(* CoDeSys 2.3 export: CRYNKAMOGILEV.EXP *)
(* Libraries: Iecsfc.lib 30.1.13 14:05:12, Standard.lib 20.5.14 09:13:26, SYSLIBCALLBACK.LIB 30.1.13 14:05:12, SysLibRtc.lib 30.1.13 14:05:12, SysLibTime.lib 30.1.13 14:05:12, Util_no_Real.lib 30.1.13 14:05:12 *)

(* PLC configuration (modules and I/O channels)
PLC Configuration [Root] node -1, in %IB0 out %QB0
  K-Bus [K_Bus] node 0, in %IB0 out %QB0 {param 201019000 = 1; param 201019001 = 10000; param 201019002 = 0; param 201019003 = 1}
    0750-1405 16 DI 24V DC 3.0ms [Type_1_16_Channels] node 0, in %IB56 out %QB16
      _Pump_FeedbackOn_1 AT %IX28.0 [BOOLOnX_I] Ch_1 Digital input
      _Pump_Alm_1 AT %IX28.1 [BOOLOnX_I] Ch_2 Digital input
      _Pump_FeedbackOn_2 AT %IX28.2 [BOOLOnX_I] Ch_3 Digital input
      _Pump_Alm_2 AT %IX28.3 [BOOLOnX_I] Ch_4 Digital input
      _Pump_FeedbackOn_3 AT %IX28.4 [BOOLOnX_I] Ch_5 Digital input
      _Pump_Alm_3 AT %IX28.5 [BOOLOnX_I] Ch_6 Digital input
      _Pump_FeedbackOn_4 AT %IX28.6 [BOOLOnX_I] Ch_7 Digital input
      _Pump_Alm_4 AT %IX28.7 [BOOLOnX_I] Ch_8 Digital input
      _DI_FeedBackSwitchLine1 AT %IX28.8 [BOOLOnX_I] Ch_9 Digital input
      _DI_FeedBackSwitchLine2 AT %IX28.9 [BOOLOnX_I] Ch_10 Digital input
      _DI_FeedBackSwitchLine3 AT %IX28.10 [BOOLOnX_I] Ch_11 Digital input
      _DI_FeedBackSwitchLine4 AT %IX28.11 [BOOLOnX_I] Ch_12 Digital input
      _LH_1 AT %IX28.12 [BOOLOnX_I] Ch_13 Digital input
      _LH_2 AT %IX28.13 [BOOLOnX_I] Ch_14 Digital input
      _LH_3 AT %IX28.14 [BOOLOnX_I] Ch_15 Digital input
      _LH_4 AT %IX28.15 [BOOLOnX_I] Ch_16 Digital input
    0750-1405 16 DI 24V DC 3.0ms [Type_1_16_Channels] node 1, in %IB56 out %QB16
      _FC_1 AT %IX29.0 [BOOLOnX_I] Ch_1 Digital input
      _FC_2 AT %IX29.1 [BOOLOnX_I] Ch_2 Digital input
      _FC_3 AT %IX29.2 [BOOLOnX_I] Ch_3 Digital input
      _FC_4 AT %IX29.3 [BOOLOnX_I] Ch_4 Digital input
      _Permition_Line_1 AT %IX29.4 [BOOLOnX_I] Ch_5 Digital input
      _Permition_Line_2 AT %IX29.5 [BOOLOnX_I] Ch_6 Digital input
      _Permition_Line_3 AT %IX29.6 [BOOLOnX_I] Ch_7 Digital input
      _Permition_Line_4 AT %IX29.7 [BOOLOnX_I] Ch_8 Digital input
      _Permition_Line_5 AT %IX29.8 [BOOLOnX_I] Ch_9 Digital input
      AT %IX29.9 [BOOLOnX_I] Ch_10 Digital input
      AT %IX29.10 [BOOLOnX_I] Ch_11 Digital input
      AT %IX29.11 [BOOLOnX_I] Ch_12 Digital input
      AT %IX29.12 [BOOLOnX_I] Ch_13 Digital input
      AT %IX29.13 [BOOLOnX_I] Ch_14 Digital input
      AT %IX29.14 [BOOLOnX_I] Ch_15 Digital input
      AT %IX29.15 [BOOLOnX_I] Ch_16 Digital input
    0750-1405 16 DI 24V DC 3.0ms [Type_1_16_Channels] node 2, in %IB58 out %QB16
      AT %IX30.0 [BOOLOnX_I] Ch_1 Digital input
      AT %IX30.1 [BOOLOnX_I] Ch_2 Digital input
      AT %IX30.2 [BOOLOnX_I] Ch_3 Digital input
      AT %IX30.3 [BOOLOnX_I] Ch_4 Digital input
      AT %IX30.4 [BOOLOnX_I] Ch_5 Digital input
      AT %IX30.5 [BOOLOnX_I] Ch_6 Digital input
      AT %IX30.6 [BOOLOnX_I] Ch_7 Digital input
      AT %IX30.7 [BOOLOnX_I] Ch_8 Digital input
      _DI_V101 AT %IX30.8 [BOOLOnX_I] Ch_9 Digital input
      _DI_V102 AT %IX30.9 [BOOLOnX_I] Ch_10 Digital input
      _DI_V103 AT %IX30.10 [BOOLOnX_I] Ch_11 Digital input
      _DI_V104 AT %IX30.11 [BOOLOnX_I] Ch_12 Digital input
      _DI_V105 AT %IX30.12 [BOOLOnX_I] Ch_13 Digital input
      _DI_V106 AT %IX30.13 [BOOLOnX_I] Ch_14 Digital input
      _DI_V107 AT %IX30.14 [BOOLOnX_I] Ch_15 Digital input
      _DI_V108 AT %IX30.15 [BOOLOnX_I] Ch_16 Digital input
    0750-1405 16 DI 24V DC 3.0ms [Type_1_16_Channels] node 3, in %IB60 out %QB16
      _DI_V109 AT %IX31.0 [BOOLOnX_I] Ch_1 Digital input
      _DI_V110 AT %IX31.1 [BOOLOnX_I] Ch_2 Digital input
      _DI_V111 AT %IX31.2 [BOOLOnX_I] Ch_3 Digital input
      _DI_V201 AT %IX31.3 [BOOLOnX_I] Ch_4 Digital input
      _DI_V202 AT %IX31.4 [BOOLOnX_I] Ch_5 Digital input
      _DI_V203 AT %IX31.5 [BOOLOnX_I] Ch_6 Digital input
      _DI_V204 AT %IX31.6 [BOOLOnX_I] Ch_7 Digital input
      _DI_V205 AT %IX31.7 [BOOLOnX_I] Ch_8 Digital input
      _DI_V206 AT %IX31.8 [BOOLOnX_I] Ch_9 Digital input
      _DI_V207 AT %IX31.9 [BOOLOnX_I] Ch_10 Digital input
      _DI_V208 AT %IX31.10 [BOOLOnX_I] Ch_11 Digital input
      _DI_V209 AT %IX31.11 [BOOLOnX_I] Ch_12 Digital input
      _DI_V210 AT %IX31.12 [BOOLOnX_I] Ch_13 Digital input
      _DI_V211 AT %IX31.13 [BOOLOnX_I] Ch_14 Digital input
      _DI_V301 AT %IX31.14 [BOOLOnX_I] Ch_15 Digital input
      _DI_V302 AT %IX31.15 [BOOLOnX_I] Ch_16 Digital input
    0750-1405 16 DI 24V DC 3.0ms [Type_1_16_Channels] node 4, in %IB62 out %QB16
      _DI_V303 AT %IX32.0 [BOOLOnX_I] Ch_1 Digital input
      _DI_V304 AT %IX32.1 [BOOLOnX_I] Ch_2 Digital input
      _DI_V305 AT %IX32.2 [BOOLOnX_I] Ch_3 Digital input
      _DI_V306 AT %IX32.3 [BOOLOnX_I] Ch_4 Digital input
      _DI_V307 AT %IX32.4 [BOOLOnX_I] Ch_5 Digital input
      _DI_V308 AT %IX32.5 [BOOLOnX_I] Ch_6 Digital input
      _DI_V309 AT %IX32.6 [BOOLOnX_I] Ch_7 Digital input
      _DI_V310 AT %IX32.7 [BOOLOnX_I] Ch_8 Digital input
      _DI_V311 AT %IX32.8 [BOOLOnX_I] Ch_9 Digital input
      _DI_V401 AT %IX32.9 [BOOLOnX_I] Ch_10 Digital input
      _DI_V402 AT %IX32.10 [BOOLOnX_I] Ch_11 Digital input
      _DI_V403 AT %IX32.11 [BOOLOnX_I] Ch_12 Digital input
      _DI_V404 AT %IX32.12 [BOOLOnX_I] Ch_13 Digital input
      _DI_V405 AT %IX32.13 [BOOLOnX_I] Ch_14 Digital input
      _DI_V406 AT %IX32.14 [BOOLOnX_I] Ch_15 Digital input
      _DI_V407 AT %IX32.15 [BOOLOnX_I] Ch_16 Digital input
    0750-1405 16 DI 24V DC 3.0ms [Type_1_16_Channels] node 5, in %IB64 out %QB16
      _DI_V408 AT %IX33.0 [BOOLOnX_I] Ch_1 Digital input
      _DI_V409 AT %IX33.1 [BOOLOnX_I] Ch_2 Digital input
      _DI_V410 AT %IX33.2 [BOOLOnX_I] Ch_3 Digital input
      _DI_V411 AT %IX33.3 [BOOLOnX_I] Ch_4 Digital input
      _DI_V510 AT %IX33.4 [BOOLOnX_I] Ch_5 Digital input
      _DI_V511 AT %IX33.5 [BOOLOnX_I] Ch_6 Digital input
      _DI_V512 AT %IX33.6 [BOOLOnX_I] Ch_7 Digital input
      _DI_V513 AT %IX33.7 [BOOLOnX_I] Ch_8 Digital input
      _DI_V514 AT %IX33.8 [BOOLOnX_I] Ch_9 Digital input
      _DI_V515 AT %IX33.9 [BOOLOnX_I] Ch_10 Digital input
      _DI_V501 AT %IX33.10 [BOOLOnX_I] Ch_11 Digital input
      AT %IX33.11 [BOOLOnX_I] Ch_12 Digital input
      AT %IX33.12 [BOOLOnX_I] Ch_13 Digital input
      AT %IX33.13 [BOOLOnX_I] Ch_14 Digital input
      AT %IX33.14 [BOOLOnX_I] Ch_15 Digital input
      AT %IX33.15 [BOOLOnX_I] Ch_16 Digital input
    0750-1504 16 DO 24V DC 0.5A [Type_10_16_Channels] node 6, in %IB66 out %QB16
      _DO_PumpOn_1 AT %QX8.0 [BOOLOnX_Q] Ch_1 Digital output
      _DO_PumpOn_2 AT %QX8.1 [BOOLOnX_Q] Ch_2 Digital output
      _DO_PumpOn_3 AT %QX8.2 [BOOLOnX_Q] Ch_3 Digital output
      _DO_PumpOn_4 AT %QX8.3 [BOOLOnX_Q] Ch_4 Digital output
      _HL_Green AT %QX8.4 [BOOLOnX_Q] Ch_5 Digital output
      _HL_Yellow AT %QX8.5 [BOOLOnX_Q] Ch_6 Digital output
      _HL_Red AT %QX8.6 [BOOLOnX_Q] Ch_7 Digital output
      _Alm AT %QX8.7 [BOOLOnX_Q] Ch_8 Digital output
      _Ready_Line_1 AT %QX8.8 [BOOLOnX_Q] Ch_9 Digital output
      _Working_Line_1 AT %QX8.9 [BOOLOnX_Q] Ch_10 Digital output
      _Working_Pump_1 AT %QX8.10 [BOOLOnX_Q] Ch_11 Digital output
      _SwitchOnRemotePump_1 AT %QX8.11 [BOOLOnX_Q] Ch_12 Digital output
      _SwitchOnRemotePump_2 AT %QX8.12 [BOOLOnX_Q] Ch_13 Digital output
      _Ready_Line_2 AT %QX8.13 [BOOLOnX_Q] Ch_14 Digital output
      _Working_Line_2 AT %QX8.14 [BOOLOnX_Q] Ch_15 Digital output
      _Working_Pump_2 AT %QX8.15 [BOOLOnX_Q] Ch_16 Digital output
    0750-1504 16 DO 24V DC 0.5A [Type_10_16_Channels] node 7, in %IB68 out %QB16
      AT %QX9.0 [BOOLOnX_Q] Ch_1 Digital output
      AT %QX9.1 [BOOLOnX_Q] Ch_2 Digital output
      _Ready_Line_3 AT %QX9.2 [BOOLOnX_Q] Ch_3 Digital output
      _Working_Line_3 AT %QX9.3 [BOOLOnX_Q] Ch_4 Digital output
      _Working_Pump_3 AT %QX9.4 [BOOLOnX_Q] Ch_5 Digital output
      _SwitchOnRemotePump_3 AT %QX9.5 [BOOLOnX_Q] Ch_6 Digital output
      AT %QX9.6 [BOOLOnX_Q] Ch_7 Digital output
      _Ready_Line_4 AT %QX9.7 [BOOLOnX_Q] Ch_8 Digital output
      _Working_Line_4 AT %QX9.8 [BOOLOnX_Q] Ch_9 Digital output
      _Working_Pump_4 AT %QX9.9 [BOOLOnX_Q] Ch_10 Digital output
      _SwitchOnRemotePump_4 AT %QX9.10 [BOOLOnX_Q] Ch_11 Digital output
      AT %QX9.11 [BOOLOnX_Q] Ch_12 Digital output
      AT %QX9.12 [BOOLOnX_Q] Ch_13 Digital output
      AT %QX9.13 [BOOLOnX_Q] Ch_14 Digital output
      AT %QX9.14 [BOOLOnX_Q] Ch_15 Digital output
      AT %QX9.15 [BOOLOnX_Q] Ch_16 Digital output
    0750-1504 16 DO 24V DC 0.5A [Type_10_16_Channels] node 8, in %IB68 out %QB18
      _DO_V101 AT %QX10.0 [BOOLOnX_Q] Ch_1 Digital output
      _DO_V102 AT %QX10.1 [BOOLOnX_Q] Ch_2 Digital output
      _DO_V103 AT %QX10.2 [BOOLOnX_Q] Ch_3 Digital output
      _DO_V104 AT %QX10.3 [BOOLOnX_Q] Ch_4 Digital output
      _DO_V105 AT %QX10.4 [BOOLOnX_Q] Ch_5 Digital output
      _DO_V106 AT %QX10.5 [BOOLOnX_Q] Ch_6 Digital output
      _DO_V107 AT %QX10.6 [BOOLOnX_Q] Ch_7 Digital output
      _DO_V108 AT %QX10.7 [BOOLOnX_Q] Ch_8 Digital output
      _DO_V109 AT %QX10.8 [BOOLOnX_Q] Ch_9 Digital output
      _DO_V110 AT %QX10.9 [BOOLOnX_Q] Ch_10 Digital output
      _DO_V111 AT %QX10.10 [BOOLOnX_Q] Ch_11 Digital output
      _DO_V201 AT %QX10.11 [BOOLOnX_Q] Ch_12 Digital output
      _DO_V202 AT %QX10.12 [BOOLOnX_Q] Ch_13 Digital output
      _DO_V203 AT %QX10.13 [BOOLOnX_Q] Ch_14 Digital output
      _DO_V204 AT %QX10.14 [BOOLOnX_Q] Ch_15 Digital output
      _DO_V205 AT %QX10.15 [BOOLOnX_Q] Ch_16 Digital output
    0750-1504 16 DO 24V DC 0.5A [Type_10_16_Channels] node 9, in %IB68 out %QB20
      _DO_V206 AT %QX11.0 [BOOLOnX_Q] Ch_1 Digital output
      _DO_V207 AT %QX11.1 [BOOLOnX_Q] Ch_2 Digital output
      _DO_V208 AT %QX11.2 [BOOLOnX_Q] Ch_3 Digital output
      _DO_V209 AT %QX11.3 [BOOLOnX_Q] Ch_4 Digital output
      _DO_V210 AT %QX11.4 [BOOLOnX_Q] Ch_5 Digital output
      _DO_V211 AT %QX11.5 [BOOLOnX_Q] Ch_6 Digital output
      _DO_V301 AT %QX11.6 [BOOLOnX_Q] Ch_7 Digital output
      _DO_V302 AT %QX11.7 [BOOLOnX_Q] Ch_8 Digital output
      _DO_V303 AT %QX11.8 [BOOLOnX_Q] Ch_9 Digital output
      _DO_V304 AT %QX11.9 [BOOLOnX_Q] Ch_10 Digital output
      _DO_V305 AT %QX11.10 [BOOLOnX_Q] Ch_11 Digital output
      _DO_V306 AT %QX11.11 [BOOLOnX_Q] Ch_12 Digital output
      AT %QX11.12 [BOOLOnX_Q] Ch_13 Digital output
      _DO_PA1 AT %QX11.13 [BOOLOnX_Q] Ch_14 Digital output
      _DO_PA2 AT %QX11.14 [BOOLOnX_Q] Ch_15 Digital output
      _DO_PA3 AT %QX11.15 [BOOLOnX_Q] Ch_16 Digital output
    0750-1504 16 DO 24V DC 0.5A [Type_10_16_Channels] node 10, in %IB68 out %QB22
      _DO_V308 AT %QX12.0 [BOOLOnX_Q] Ch_1 Digital output
      _DO_V309 AT %QX12.1 [BOOLOnX_Q] Ch_2 Digital output
      _DO_V310 AT %QX12.2 [BOOLOnX_Q] Ch_3 Digital output
      _DO_V311 AT %QX12.3 [BOOLOnX_Q] Ch_4 Digital output
      _DO_V401 AT %QX12.4 [BOOLOnX_Q] Ch_5 Digital output
      _DO_V402 AT %QX12.5 [BOOLOnX_Q] Ch_6 Digital output
      _DO_V403 AT %QX12.6 [BOOLOnX_Q] Ch_7 Digital output
      _DO_V404 AT %QX12.7 [BOOLOnX_Q] Ch_8 Digital output
      _DO_V405 AT %QX12.8 [BOOLOnX_Q] Ch_9 Digital output
      _DO_V406 AT %QX12.9 [BOOLOnX_Q] Ch_10 Digital output
      _DO_V407 AT %QX12.10 [BOOLOnX_Q] Ch_11 Digital output
      _DO_V408 AT %QX12.11 [BOOLOnX_Q] Ch_12 Digital output
      _DO_V409 AT %QX12.12 [BOOLOnX_Q] Ch_13 Digital output
      _DO_V410 AT %QX12.13 [BOOLOnX_Q] Ch_14 Digital output
      _DO_V411 AT %QX12.14 [BOOLOnX_Q] Ch_15 Digital output
      _DO_V510 AT %QX12.15 [BOOLOnX_Q] Ch_16 Digital output
    0750-1504 16 DO 24V DC 0.5A [Type_10_16_Channels] node 11, in %IB68 out %QB24
      _DO_V511 AT %QX13.0 [BOOLOnX_Q] Ch_1 Digital output
      _DO_V512 AT %QX13.1 [BOOLOnX_Q] Ch_2 Digital output
      _DO_V513 AT %QX13.2 [BOOLOnX_Q] Ch_3 Digital output
      _DO_V514 AT %QX13.3 [BOOLOnX_Q] Ch_4 Digital output
      _DO_V515 AT %QX13.4 [BOOLOnX_Q] Ch_5 Digital output
      _DO_V501 AT %QX13.5 [BOOLOnX_Q] Ch_6 Digital output
      _DO_V307 AT %QX13.6 [BOOLOnX_Q] Ch_7 Digital output
      AT %QX13.7 [BOOLOnX_Q] Ch_8 Digital output
      AT %QX13.8 [BOOLOnX_Q] Ch_9 Digital output
      AT %QX13.9 [BOOLOnX_Q] Ch_10 Digital output
      AT %QX13.10 [BOOLOnX_Q] Ch_11 Digital output
      AT %QX13.11 [BOOLOnX_Q] Ch_12 Digital output
      _DO_PA4 AT %QX13.12 [BOOLOnX_Q] Ch_13 Digital output
      _DO_PA11 AT %QX13.13 [BOOLOnX_Q] Ch_14 Digital output
      _DO_PA12 AT %QX13.14 [BOOLOnX_Q] Ch_15 Digital output
      AT %QX13.15 [BOOLOnX_Q] Ch_16 Digital output
    0750-0496 8AI 0-20mA/4-20mA S.E. [Type_63_8_Channels] node 12, in %IB56 out %QB8
      _AI_Conc_Line1 AT %IW0 [INTOnW_I] Ch_1 signed Input value
      _AI_Conc_Line2 AT %IW1 [INTOnW_I] Ch_2 signed Input value
      _AI_Conc_Line3 AT %IW2 [INTOnW_I] Ch_3 signed Input value
      _AI_Conc_Line4 AT %IW3 [INTOnW_I] Ch_4 signed Input value
      _AI_AccidLevel AT %IW4 [INTOnW_I] Ch_5 signed Input value
      _AI_AlkaliLevel AT %IW5 [INTOnW_I] Ch_6 signed Input value
      _AI_CleanWaterLevel AT %IW6 [INTOnW_I] Ch_7 signed Input value
      _AI_UsedWaterLevel AT %IW7 [INTOnW_I] Ch_8 signed Input value
    0750-0496 8AI 0-20mA/4-20mA S.E. [Type_63_8_Channels] node 13, in %IB56 out %QB8
      _AI_Flaw_Line1 AT %IW8 [INTOnW_I] Ch_1 signed Input value
      _AI_Flaw_Line2 AT %IW9 [INTOnW_I] Ch_2 signed Input value
      _AI_Flaw_Line3 AT %IW10 [INTOnW_I] Ch_3 signed Input value
      _AI_Flaw_Line4 AT %IW11 [INTOnW_I] Ch_4 signed Input value
      AT %IW12 [INTOnW_I] Ch_5 signed Input value
      AT %IW13 [INTOnW_I] Ch_6 signed Input value
      AT %IW14 [INTOnW_I] Ch_7 signed Input value
      AT %IW15 [INTOnW_I] Ch_8 signed Input value
    0750-0450 4AI RTD/ adj. [Type_62_4_Channels] node 14, in %IB72 out %QB8
      _AI_Heater_BackTget_1 AT %IW16 [INTOnW_I] Ch_1 signed Input value
      _AI_Heater_BackTget_2 AT %IW17 [INTOnW_I] Ch_2 signed Input value
      _AI_Heater_BackTget_3 AT %IW18 [INTOnW_I] Ch_3 signed Input value
      _AI_Heater_BackTget_4 AT %IW19 [INTOnW_I] Ch_4 signed Input value
    0750-0450 4AI RTD/ adj. [Type_62_4_Channels] node 15, in %IB88 out %QB8
      _AI_Heater_Tget_1 AT %IW20 [INTOnW_I] Ch_1 signed Input value
      _AI_Heater_Tget_2 AT %IW21 [INTOnW_I] Ch_2 signed Input value
      _AI_Heater_Tget_3 AT %IW22 [INTOnW_I] Ch_3 signed Input value
      _AI_Heater_Tget_4 AT %IW23 [INTOnW_I] Ch_4 signed Input value
    0750-0450 4AI RTD/ adj. [Type_62_4_Channels] node 16, in %IB96 out %QB8
      _AI_Temp_Accid AT %IW24 [INTOnW_I] Ch_1 signed Input value
      _AI_Temp_Alkali AT %IW25 [INTOnW_I] Ch_2 signed Input value
      AT %IW26 [INTOnW_I] Ch_3 signed Input value
      AT %IW27 [INTOnW_I] Ch_4 signed Input value
    0750-0555 4 AO 4-20mA [Type_14_4_Channels] node 17, in %IB104 out %QB8
      _AO_PumpSpeedSet_1 AT %QW0 [WORDOnW_Q] Ch_1 Analog output
      _AO_PumpSpeedSet_2 AT %QW1 [WORDOnW_Q] Ch_2 Analog output
      _AO_PumpSpeedSet_3 AT %QW2 [WORDOnW_Q] Ch_3 Analog output
      _AO_PumpSpeedSet_4 AT %QW3 [WORDOnW_Q] Ch_4 Analog output
    0750-0555 4 AO 4-20mA [Type_14_4_Channels] node 18, in %IB112 out %QB8
      _AO_HeaterPowerSet_1 AT %QW4 [WORDOnW_Q] Ch_1 Analog output
      _AO_HeaterPowerSet_2 AT %QW5 [WORDOnW_Q] Ch_2 Analog output
      _AO_HeaterPowerSet_3 AT %QW6 [WORDOnW_Q] Ch_3 Analog output
      _AO_HeaterPowerSet_4 AT %QW7 [WORDOnW_Q] Ch_4 Analog output
  Modbus variables [PFC200MODBUS] node 1, in %IB0 out %QB0 {param 2010330101 = 1; param 2010330102 = 1; param 2010330201 = 1; param 2010330202 = 502; param 2010330203 = 600; param 2010330301 = 1; param 2010330302 = 502; param 2010330401 = 0; param 2010330402 = 1; param 2010330403 = 5000; param 2010330404 = 0; param 2010330405 = 115200; param 2010330406 = 1; param 2010330407 = 1; param 2010330408 = 0; param 2010330409 = 0}
  Modbus-Master [MB_MASTER] node 2, in %IB0 out %QB0
*)

(* Global variable list: AI_Vars *)
VAR_GLOBAL

	AI_Conc_Line1:			WORD;
	AI_Conc_Line2:			WORD;
	AI_Conc_Line3:			WORD;
	AI_Conc_Line4:			WORD;

	AI_CleanWaterLevel:		WORD;
	AI_UsedWaterLevel:		WORD;
	AI_AccidLevel:				WORD;
	AI_AlkaliLevel:				WORD;

	AI_Temp_Accid:			WORD;
	AI_Temp_Alkali:			WORD;
	AI_Temp_Line3:			WORD;
	AI_Temp_Line4:			WORD;

	AI_Heater_Tget_1 	:	WORD;
	AI_Heater_Tget_2 	:	WORD;
	AI_Heater_Tget_3 	:	WORD;
	AI_Heater_Tget_4 	:	WORD;
			
	AI_Heater_BackTget_1	:	WORD;
	AI_Heater_BackTget_2	:	WORD;
	AI_Heater_BackTget_3	:	WORD;
	AI_Heater_BackTget_4	:	WORD;



	AI_Flaw_Line1:			WORD;
	AI_Flaw_Line2:			WORD;
	AI_Flaw_Line3:			WORD;
	AI_Flaw_Line4:			WORD;



END_VAR

(* Global variable list: AO_Vars *)
VAR_GLOBAL


	AO_PumpSpeedSet_1:			WORD;
	AO_PumpSpeedSet_2:			WORD;
	AO_PumpSpeedSet_3:			WORD;
	AO_PumpSpeedSet_4:			WORD;

	AO_HeaterPowerSet_1 AT %MW1060:			WORD;
	AO_HeaterPowerSet_2 AT %MW1062:			WORD;
	AO_HeaterPowerSet_3 AT %MW1064:			WORD;
	AO_HeaterPowerSet_4 AT %MW1066:			WORD;
END_VAR

(* Global variable list: DI_Vars *)
VAR_GLOBAL



	DI_V101	:	BOOL;
	DI_V102	:	BOOL;
	DI_V103	:	BOOL;
	DI_V104	:	BOOL;
	DI_V105	:	BOOL;
	DI_V106	:	BOOL;
	DI_V107	:	BOOL;
	DI_V108	:	BOOL;
	DI_V109	:	BOOL;
	DI_V110	:	BOOL;
	DI_V111	:	BOOL;
	DI_V201	:	BOOL;
	DI_V202	:	BOOL;
	DI_V203	:	BOOL;
	DI_V204	:	BOOL;
	DI_V205	:	BOOL;
	DI_V206	:	BOOL;
	DI_V207	:	BOOL;
	DI_V208	:	BOOL;
	DI_V209	:	BOOL;
	DI_V210	:	BOOL;
	DI_V211	:	BOOL;
	DI_V301	:	BOOL;
	DI_V302	:	BOOL;
	DI_V303	:	BOOL;
	DI_V304	:	BOOL;
	DI_V305	:	BOOL;
	DI_V306	:	BOOL;
	DI_V307	:	BOOL;
	DI_V308	:	BOOL;
	DI_V309	:	BOOL;
	DI_V310	:	BOOL;
	DI_V311	:	BOOL;
	DI_V401	:	BOOL;
	DI_V402	:	BOOL;
	DI_V403	:	BOOL;
	DI_V404	:	BOOL;
	DI_V405	:	BOOL;
	DI_V406	:	BOOL;
	DI_V407	:	BOOL;
	DI_V408	:	BOOL;
	DI_V409	:	BOOL;
	DI_V410	:	BOOL;
	DI_V411	:	BOOL;
	DI_V501	:	BOOL;
	DI_V510	:	BOOL;
	DI_V511	:	BOOL;
	DI_V512	:	BOOL;
	DI_V513	:	BOOL;
	DI_V514	:	BOOL;
	DI_V515	:	BOOL;


	Pump_InvNorm_1:	BOOL;
	Pump_InvNorm_2:	BOOL;
	Pump_InvNorm_3:	BOOL;
	Pump_InvNorm_4:	BOOL;

	Permition_Line_1:	BOOL;
	Permition_Line_2:	BOOL;
	Permition_Line_3:	BOOL;
	Permition_Line_4:	BOOL;
	Permition_Line_5:	BOOL;





END_VAR

(* Global variable list: DO_Vars *)
VAR_GLOBAL
	DO_PumpOn_1:			BOOL;
	DO_PumpOn_2:			BOOL;
	DO_PumpOn_3:			BOOL;
	DO_PumpOn_4:			BOOL;

	DO_PA11:					BOOL;
	DO_PA12:					BOOL;
	DO_PA1:					BOOL;
	DO_PA2:					BOOL;
	DO_PA3:					BOOL;
	DO_PA4:					BOOL;

	DO_V110	:	BOOL;
	DO_V210	:	BOOL;
	DO_V310	:	BOOL;
	DO_V410	:	BOOL;
	DO_V111	:	BOOL;
	DO_V211	:	BOOL;
	DO_V311	:	BOOL;
	DO_V411	:	BOOL;
			
	DO_V101	:	BOOL;
	DO_V102	:	BOOL;
	DO_V103	:	BOOL;
	DO_V104	:	BOOL;
	DO_V105	:	BOOL;
	DO_V106	:	BOOL;
	DO_V107	:	BOOL;
	DO_V108	:	BOOL;
	DO_V109	:	BOOL;
	DO_V201	:	BOOL;
	DO_V202	:	BOOL;
	DO_V203	:	BOOL;
	DO_V204	:	BOOL;
	DO_V205	:	BOOL;
	DO_V206	:	BOOL;
	DO_V207	:	BOOL;
	DO_V208	:	BOOL;
	DO_V209	:	BOOL;
	DO_V301	:	BOOL;
	DO_V302	:	BOOL;
	DO_V303	:	BOOL;
	DO_V304	:	BOOL;
	DO_V305	:	BOOL;
	DO_V306	:	BOOL;
	DO_V307	:	BOOL;
	DO_V308	:	BOOL;
	DO_V309	:	BOOL;
	DO_V401	:	BOOL;
	DO_V402	:	BOOL;
	DO_V403	:	BOOL;
	DO_V404	:	BOOL;
	DO_V405	:	BOOL;
	DO_V406	:	BOOL;
	DO_V407	:	BOOL;
	DO_V408	:	BOOL;
	DO_V409	:	BOOL;
		
	DO_V501	:	BOOL;
		
	DO_V511	:	BOOL;
	DO_V510	:	BOOL;
	DO_V512	:	BOOL;
	DO_V513	:	BOOL;
	DO_V514	:	BOOL;
	DO_V515	:	BOOL;

	DO_ReadyToWash:					BOOL;
	DO_WashimgIsGoing:				BOOL;
	DO_PumpIsWorking:					BOOL;

	SwitchOnRemotePump_1	:	BOOL;
	SwitchOnRemotePump_2	:	BOOL;
	SwitchOnRemotePump_3	:	BOOL;
	SwitchOnRemotePump_4	:	BOOL;

	SwitchOnRemotePump_1_1	:	BOOL;
	SwitchOnRemotePump_1_2	:	BOOL;
	SwitchOnRemotePump_1_3	:	BOOL;


END_VAR

(* Global variable list: Global_Variables *)
VAR_GLOBAL
	Bob: BOOL;
	Seed: WORD;
	ffggh:WORD;
	kkfggj:WORD;
	xReadyForWashing:	BOOL;

END_VAR

(* Global variable list: Heater *)
VAR_GLOBAL

	Heater_AutoSetT_1:					REAL;
	Heater_AutoSetT_2:					REAL;
	Heater_AutoSetT_3:					REAL;
	Heater_AutoSetT_4:					REAL;

END_VAR

(* Global variable list: HMI_Alarms *)
VAR_GLOBAL

	xResetAlmAll	AT %MW600	:	BOOL;	(*	12888	*)
						
	wAlm_V101	AT %MW601	:	WORD;	(*	12889	*)
	wAlm_V102	AT %MW602	:	WORD;	(*	12890	*)
	wAlm_V103	AT %MW603	:	WORD;	(*	12891	*)
	wAlm_V104	AT %MW604	:	WORD;	(*	12892	*)
	wAlm_V105	AT %MW605	:	WORD;	(*	12893	*)
	wAlm_V106	AT %MW606	:	WORD;	(*	12894	*)
	wAlm_V107	AT %MW607	:	WORD;	(*	12895	*)
	wAlm_V108	AT %MW608	:	WORD;	(*	12896	*)
	wAlm_V109	AT %MW609	:	WORD;	(*	12897	*)
	wAlm_V110	AT %MW610	:	WORD;	(*	12898	*)
	wAlm_V111	AT %MW611	:	WORD;	(*	12899	*)
	wAlm_V201	AT %MW612	:	WORD;	(*	12900	*)
	wAlm_V202	AT %MW613	:	WORD;	(*	12901	*)
	wAlm_V203	AT %MW614	:	WORD;	(*	12902	*)
	wAlm_V204	AT %MW615	:	WORD;	(*	12903	*)
	wAlm_V205	AT %MW616	:	WORD;	(*	12904	*)
	wAlm_V206	AT %MW617	:	WORD;	(*	12905	*)
	wAlm_V207	AT %MW618	:	WORD;	(*	12906	*)
	wAlm_V208	AT %MW619	:	WORD;	(*	12907	*)
	wAlm_V209	AT %MW620	:	WORD;	(*	12908	*)
	wAlm_V210	AT %MW621	:	WORD;	(*	12909	*)
	wAlm_V211	AT %MW622	:	WORD;	(*	12910	*)
	wAlm_V301	AT %MW623	:	WORD;	(*	12911	*)
	wAlm_V302	AT %MW624	:	WORD;	(*	12912	*)
	wAlm_V303	AT %MW625	:	WORD;	(*	12913	*)
	wAlm_V304	AT %MW626	:	WORD;	(*	12914	*)
	wAlm_V305	AT %MW627	:	WORD;	(*	12915	*)
	wAlm_V306	AT %MW628	:	WORD;	(*	12916	*)
	wAlm_V307	AT %MW629	:	WORD;	(*	12917	*)
	wAlm_V308	AT %MW630	:	WORD;	(*	12918	*)
	wAlm_V309	AT %MW631	:	WORD;	(*	12919	*)
	wAlm_V310	AT %MW632	:	WORD;	(*	12920	*)
	wAlm_V311	AT %MW633	:	WORD;	(*	12921	*)
	wAlm_V401	AT %MW634	:	WORD;	(*	12922	*)
	wAlm_V402	AT %MW635	:	WORD;	(*	12923	*)
	wAlm_V403	AT %MW636	:	WORD;	(*	12924	*)
	wAlm_V404	AT %MW637	:	WORD;	(*	12925	*)
	wAlm_V405	AT %MW638	:	WORD;	(*	12926	*)
	wAlm_V406	AT %MW639	:	WORD;	(*	12927	*)
	wAlm_V407	AT %MW640	:	WORD;	(*	12928	*)
	wAlm_V408	AT %MW641	:	WORD;	(*	12929	*)
	wAlm_V409	AT %MW642	:	WORD;	(*	12930	*)
	wAlm_V410	AT %MW643	:	WORD;	(*	12931	*)
	wAlm_V411	AT %MW644	:	WORD;	(*	12932	*)
	wAlm_V501	AT %MW645	:	WORD;	(*	12933	*)
	wAlm_V510	AT %MW646	:	WORD;	(*	12934	*)
	wAlm_V511	AT %MW647	:	WORD;	(*	12935	*)
	wAlm_V512	AT %MW648	:	WORD;	(*	12936	*)
	wAlm_V513	AT %MW649	:	WORD;	(*	12937	*)
	wAlm_V514	AT %MW650	:	WORD;	(*	12938	*)
	wAlm_V515	AT %MW651	:	WORD;	(*	12939	*)
							
	wCheckAlm:			WORD;			




END_VAR

(* Global variable list: HMI_Heater *)
VAR_GLOBAL

	Heater_Tget_1 				AT %MW100:		REAL;	(* 12388 *)
	Heater_Tget_2 				AT %MW102:		REAL;	(* 12390 *)
	Heater_Tget_3 				AT %MW104:		REAL;	(* 12392 *)
	Heater_Tget_4 				AT %MW106:		REAL;	(* 12394 *)

	Heater_Error_1 				AT %MW108:		WORD; (* 12396 *)
	Heater_Error_2 				AT %MW110:		WORD; (* 12398 *)
	Heater_Error_3 				AT %MW112:		WORD; (* 12400 *)
	Heater_Error_4 				AT %MW114:		WORD; (* 12402 *)

	Heater_xNoFeedback_1		AT %MW116:		BOOL;	(* 12404 *)
	Heater_xNoFeedback_2 		AT %MW118:	  	BOOL;	(* 12406 *)
	Heater_xNoFeedback_3 		AT %MW120:		BOOL;	(* 12408 *)
	Heater_xNoFeedback_4 		AT %MW122:		BOOL;	(* 12410 *)

	Heater_ManualSetT_1 		AT %MW124:		REAL;	(* 12412 *)
	Heater_ManualSetT_2 		AT %MW126:		REAL;	(* 12414 *)
	Heater_ManualSetT_3 		AT %MW128:	  	REAL;	(* 12416 *)
	Heater_ManualSetT_4		AT %MW130:		REAL;	(* 12418 *)

	Heater_PowerSet_1 			AT %MW132:		REAL;	(* 12420 *)
	Heater_PowerSet_2 			AT %MW134:		REAL;	(* 12422 *)
	Heater_PowerSet_3 			AT %MW136:		REAL;	(* 12424 *)
	Heater_PowerSet_4 			AT %MW138:		REAL;	(* 12426 *)

	HeaterPowerSet_1	AT %MW140	:	REAL;	(*	12428	*)
	HeaterPowerSet_2	AT %MW142	:	REAL;	(*	12430	*)
	HeaterPowerSet_3	AT %MW144	:	REAL;	(*	12432	*)
	HeaterPowerSet_4	AT %MW146	:	REAL;	(*	12432	*)

	Heater_BackTget_1	AT %MW148	:	REAL;	(*	12434	*)
	Heater_BackTget_2	AT %MW150	:	REAL;	(*	12436	*)
	Heater_BackTget_3	AT %MW152	:	REAL;	(*	12438	*)
	Heater_BackTget_4	AT %MW154	:	REAL;	(*	12440	*)




END_VAR

VAR_GLOBAL RETAIN



	Heater_xManualMode_1		AT %MW1140	:			BOOL; 	(*	13428	*)
	Heater_xManualMode_2		AT %MW1142	:			BOOL; 	(*	13430	*)
	Heater_xManualMode_3		AT %MW1144	:			BOOL; 	(*	13432	*)
	Heater_xManualMode_4		AT %MW1146	:			BOOL; 	(*	13434	*)
END_VAR

(* Global variable list: HMI_Process *)
VAR_GLOBAL


	xDissolving_Pause			AT %MW199:		BOOL;	(* 12487 *)
	xResetErrorAll 				AT %MW200:		BOOL;	(* 12488 *)
	xDissolving_Start 				AT %MW201:		BOOL;	(* 12489 *)
	xDissolving_Stop 				AT %MW202:		BOOL;	(* 12490 *)




	xStartDissolvingAlkali		AT %MW232	:	BOOL;	(*	12520	*)
	xStartDissolvingAccid		AT %MW233	:	BOOL;	(*	12521	*)
	xPauseDissolvingAlkali	AT %MW234	:	BOOL;	(*	12522	*)
	xPauseDissolvingAccid	AT %MW235	:	BOOL;	(*	12523	*)

	wChosenRecipeLine1 		AT %MW203:		WORD:=1;(* 12491 *)
	wChosenRecipeLine2 		AT %MW204:		WORD:=1;(* 12492 *)
	wChosenRecipeLine3 		AT %MW205:		WORD:=1;(* 12493 *)
	wChosenRecipeLine4 		AT %MW206:		WORD:=1;(* 12494 *)

	wDissolvingStateLine1 		AT %MW207:		WORD;(* 12495 *)
	wDissolvingStateLine2 		AT %MW208:		WORD;(* 12496 *)
	wDissolvingStateLine3 		AT %MW209:		WORD;(* 12497 *)
	wDissolvingStateLine4 		AT %MW210:		WORD;(* 12498 *)

	wDissolvingPauseStateLine1		AT %MW236	:	WORD;	(*	12524	*)
	wDissolvingPauseStateLine2		AT %MW237	:	WORD;	(*	12525	*)
	wDissolvingPauseStateLine3		AT %MW238	:	WORD;	(*	12526	*)
	wDissolvingPauseStateLine4		AT %MW239	:	WORD;	(*	12527	*)

	wDissolvingError 				AT %MW211:		WORD;(* 12499 *)

	xStartWashingLine1 			AT %MW212:		BOOL;	(* 12500 *)
	xStartWashingLine2 			AT %MW213:		BOOL;	(* 12501 *)
	xStartWashingLine3 			AT %MW214:		BOOL;	(* 12502 *)
	xStartWashingLine4 			AT %MW215:		BOOL;	(* 12503 *)

	xPauseWashingLine1	AT %MW240	:	BOOL;	(*	12528	*)
	xPauseWashingLine2	AT %MW241	:	BOOL;	(*	12529	*)
	xPauseWashingLine3	AT %MW242	:	BOOL;	(*	12530	*)
	xPauseWashingLine4	AT %MW243	:	BOOL;	(*	12531	*)

	wWashingPauseStateLine1	AT %MW244	:	WORD;	(*	12532	*)
	wWashingPauseStateLine2	AT %MW245	:	WORD;	(*	12533	*)
	wWashingPauseStateLine3	AT %MW246	:	WORD;	(*	12534	*)
	wWashingPauseStateLine4	AT %MW247	:	WORD;	(*	12535	*)

	wWashingTimePassed1	AT %MW248	:	WORD;	(*	12536	*)
	wWashingTimePassed2	AT %MW249	:	WORD;	(*	12537	*)
	wWashingTimePassed3	AT %MW250	:	WORD;	(*	12538	*)
	wWashingTimePassed4	AT %MW251	:	WORD;	(*	12539	*)

	wWashingOperTimeSet1	AT %MW252	:	WORD;	(*	12540	*)
	wWashingOperTimeSet2	AT %MW253	:	WORD;	(*	12541	*)
	wWashingOperTimeSet3	AT %MW254	:	WORD;	(*	12542	*)
	wWashingOperTimeSet4	AT %MW255	:	WORD;	(*	12543	*)



	wWashingStateLine1 		AT %MW216:		WORD;(* 12504 *)
	wWashingStateLine2 		AT %MW217:		WORD;(* 12505 *)
	wWashingStateLine3 		AT %MW218:		WORD;(* 12506 *)
	wWashingStateLine4 		AT %MW219:		WORD;(* 12507 *)


	wWashingStateBitsLine1: 				DWORD;(* 12504 *)
	wWashingStateBitsLine2 : 				DWORD;(* 12504 *)
	wWashingStateBitsLine3 : 				DWORD;(* 12504 *)
	wWashingStateBitsLine4 : 				DWORD;(* 12504 *)

	wDissolvingStateBitsLine1 : 				DWORD;(* 12504 *)
	wDissolvingStateBitsLine2 : 				DWORD;(* 12504 *)
	wDissolvingStateBitsLine3 	: 			DWORD;(* 12504 *)
	wDissolvingStateBitsLine4 : 				DWORD;(* 12504 *)


	wWashingErr 					AT %MW220:		WORD;(* 12508 *)
	wWachingLine 				AT %MW221:		WORD;(* 12509 *)

	SelfWashDoWaterTank  			AT %MW222:		BOOL;	(* 12510 *)
	SelfWashDoUsedWaterTank  	AT %MW223:		BOOL;	(* 12511 *)
	SelfWashDoAlkaliTank  			AT %MW224:		BOOL;	(* 12512 *)
	SelfWashDoAccidTank  			AT %MW225:		BOOL;	(* 12513 *)
	SelfWashWaterIsReady  			AT %MW226:		BOOL;	(* 12514 *)
	SelfWashUsedWaterIsReady 	 AT %MW227:		BOOL;	(* 12515 *)
	SelfWashAlkaliIsReady  			AT %MW228:		BOOL;	(* 12516 *)
	SelfWashAccidIsReady  			AT %MW229:		BOOL;	(* 12517 *)
	xStartSelfWashing 				AT %MW230:		BOOL;	(* 12518 *)
	SelfWashState 					AT %MW231:		WORD;(* 12519 *)
	SelfWashStateBits:									DWORD;
	SelfWashStateBits2:									DWORD;

	xSelsWashingPause			AT %MW256	:	BOOL;		(*	12544	*)
	SelfWashPauseState			AT %MW257	:	WORD;	(*	12545	*)
	SelfWashingTimePast		AT %MW258	:	WORD;	(*	12546	*)
	SelfWashingOperTimeSet	AT %MW259	:	WORD;	(*	12547	*)
	SelfWashingAcknawlage		AT %MW260	:	BOOL;		(*	12548	*)

	wWashingErr_1	AT %MW261	:	WORD;	(*	12549	*)
	wWashingErr_2	AT %MW262	:	WORD;	(*	12550	*)
	wWashingErr_3	AT %MW263	:	WORD;	(*	12551	*)
	wWashingErr_4	AT %MW264	:	WORD;	(*	12552	*)
	xWashingDone_Line1	AT %MW1210:			BOOL;
	xWashingDone_Line2 	AT %MW1211:			BOOL;
	xWashingDone_Line3	AT %MW1212:			BOOL;
	xWashingDone_Line4	AT %MW1213:			BOOL;


END_VAR

(* Global variable list: HMI_Pump *)
VAR_GLOBAL
	Pump_FlawGet_1 			AT %MW300:		REAL;	(* 12588 *)
	Pump_FlawGet_2 			AT %MW302:		REAL;	(* 12590 *)
	Pump_FlawGet_3 			AT %MW304:		REAL;	(* 12592 *)
	Pump_FlawGet_4 			AT %MW306:		REAL;	(* 12594 *)

	Pump_OnManual_1 			AT %MW308:		BOOL;	(* 12596 *)
	Pump_OnManual_2 			AT %MW310:		BOOL;	(* 12598 *)
	Pump_OnManual_3 			AT %MW312:		BOOL;	(* 12600 *)
	Pump_OnManual_4 			AT %MW314:		BOOL;	(* 12602 *)

	Pump_NoFeedback_1 		AT %MW316:		BOOL;	(* 12604 *)
	Pump_NoFeedback_2 		AT %MW318:		BOOL;	(* 12606 *)
	Pump_NoFeedback_3 		AT %MW320:		BOOL;	(* 12608 *)
	Pump_NoFeedback_4 		AT %MW322:		BOOL;	(* 12610 *)

	Pump_Error_1 				AT %MW324:		WORD; (* 12612 *)
	Pump_Error_2 				AT %MW326:		WORD; (* 12614 *)
	Pump_Error_3 				AT %MW328:		WORD; (* 12616 *)
	Pump_Error_4 				AT %MW330:		WORD; (* 12618 *)

	Pump_OnAuto_1				AT %MW356	:	BOOL;	(*	12644	*)
	Pump_OnAuto_2				AT %MW358	:	BOOL;	(*	12646	*)
	Pump_OnAuto_3				AT %MW360	:	BOOL;	(*	12648	*)
	Pump_OnAuto_4				AT %MW362	:	BOOL;	(*	12650	*)

	Pump_BackFlawGet_1		AT %MW364	:	REAL;	(*	12652	*)
	Pump_BackFlawGet_2		AT %MW366	:	REAL;	(*	12654	*)
	Pump_BackFlawGet_3		AT %MW368	:	REAL;	(*	12656	*)
	Pump_BackFlawGet_4		AT %MW370	:	REAL;	(*	12658	*)

	PumpSpeedSet_1			AT %MW372	:	REAL;	(*	12660	*)
	PumpSpeedSet_2			AT %MW374	:	REAL;	(*	12662	*)
	PumpSpeedSet_3			AT %MW376	:	REAL;	(*	12664	*)
	PumpSpeedSet_4			AT %MW378	:	REAL;	(*	12666	*)

	Pump_FeedbackOn_1	AT %MW380	:	BOOL;	(*	12668	*)
	Pump_FeedbackOn_2	AT %MW382	:	BOOL;	(*	12670	*)
	Pump_FeedbackOn_3	AT %MW384	:	BOOL;	(*	12672	*)
	Pump_FeedbackOn_4	AT %MW386	:	BOOL;	(*	12674	*)

	PA_OnManual_1 			AT %MW388	:	BOOL;	(*	12676	*)
	PA_OnManual_2 			AT %MW390	:	BOOL;	(*	12678	*)
	PA_OnManual_3 			AT %MW392	:	BOOL;	(*	12680	*)
	PA_OnManual_4 			AT %MW394	:	BOOL;	(*	12682	*)

	PA_OnManual_11 		AT %MW396	:	BOOL;	(*	12684	*)
	PA_OnManual_12			AT %MW398	:	BOOL;	(*	12686	*)

	PA_OnAuto_1				AT %MW1000	:	BOOL;	(*	13288	*)
	PA_OnAuto_2				AT %MW1002	:	BOOL;	(*	13290	*)
	PA_OnAuto_3				AT %MW1004	:	BOOL;	(*	13292	*)
	PA_OnAuto_4				AT %MW1006	:	BOOL;	(*	13294	*)

	PA_OnAuto_11			AT %MW1008	:	BOOL;	(*	13296	*)
	PA_OnAuto_12			AT %MW1010	:	BOOL;	(*	13298	*)

	PA_State_1			AT %MW1012	:	BOOL;	(*	13300	*)
	PA_State_2			AT %MW1014	:	BOOL;	(*	13302	*)
	PA_State_3			AT %MW1016	:	BOOL;	(*	13304	*)
	PA_State_4			AT %MW1018	:	BOOL;	(*	13306	*)

	PA_State_11			AT %MW1020	:	BOOL;	(*	13308	*)
	PA_State_12			AT %MW1022	:	BOOL;	(*	13310	*)

	Pump_State_1		AT %MW1024	:	WORD;	(*	13312	*)
	Pump_State_2		AT %MW1026	:	WORD;	(*	13314	*)
	Pump_State_3		AT %MW1028	:	WORD;	(*	13316	*)
	Pump_State_4		AT %MW1030	:	WORD;	(*	13318	*)


END_VAR

VAR_GLOBAL RETAIN PERSISTENT



	Pump_ManualMode_1 		AT %MW332:		BOOL;	(* 12620 *)
	Pump_ManualMode_2 		AT %MW334:		BOOL;	(* 12622 *)
	Pump_ManualMode_3 		AT %MW336:		BOOL;	(* 12624 *)
	Pump_ManualMode_4 		AT %MW338:		BOOL;	(* 12626 *)

	Pump_FlawManualSet_1 	AT %MW340:		WORD; (* 12628 *)
	Pump_FlawManualSet_2 	AT %MW342:		WORD; (* 12630 *)
	Pump_FlawManualSet_3 	AT %MW344:		WORD; (* 12632 *)
	Pump_FlawManualSet_4 	AT %MW346:		WORD; (* 12634 *)

	Pump_VelocitySet_1 			AT %MW348:		WORD; (* 12636 *)
	Pump_VelocitySet_2 			AT %MW350:		WORD; (* 12638 *)
	Pump_VelocitySet_3 			AT %MW352:		WORD; (* 12640 *)
	Pump_VelocitySet_4 			AT %MW354:		WORD; (* 12642 *)

	PA_ManualMode_1	AT %MW1032	:	BOOL;	(*	13320	*)
	PA_ManualMode_2	AT %MW1034	:	BOOL;	(*	13322	*)
	PA_ManualMode_3	AT %MW1036	:	BOOL;	(*	13324	*)
	PA_ManualMode_4	AT %MW1038	:	BOOL;	(*	13326	*)

	PA_ManualMode_11	AT %MW1040	:	BOOL;	(*	13328	*)
	PA_ManualMode_12	AT %MW1042	:	BOOL;	(*	13330	*)

	sCheckSrting	AT %MW1050	:	WORD;	(*	13338	*)

END_VAR

(* Global variable list: HMI_Recipe *)
VAR_GLOBAL

	wLine  			AT %MW400:				WORD:=2;
	wRecipe		AT %MW402:				WORD;
	xSave			AT %MW404:				BOOL;


END_VAR
VAR_GLOBAL RETAIN PERSISTENT



	wAlkaliTime 					AT %MW406:		WORD;	(* 12694 *)
	wTalkaliSet  					AT %MW408:		WORD;	(* 12696 *)
	wFlawAlkaliSet  				AT %MW410:		REAL;	(* 12698 *)
	wConcAlkaliSet  				AT %MW412:		REAL;	(* 12700 *)
	wAccidTime 					AT %MW414:		WORD;	(* 12702 *)
	wTaccidSet  					AT %MW416:		WORD;	(* 12704 *)
	wFlawAccidSet  				AT %MW418:		REAL;	(* 12706 *)
	wConcAccidSet 				AT %MW420:		REAL;	(* 12708 *)
	wWaterTime  					AT %MW422:		WORD;	(* 12710 *)
	wTwaterSet  					AT %MW424:		WORD;	(* 12712 *)
	wFlawWaterSet  				AT %MW426:		REAL;	(* 12714 *)
	wAfterAccidWaterTime  		AT %MW428:		WORD;	(* 12716 *)
	wTafterAccidWater  			AT %MW430:		WORD;	(* 12718 *)
	wConcAfterAccidWaterSet  	AT %MW432:		REAL;	(* 12720 *)
	wAfterAlkaliWaterTime  		AT %MW434:		WORD;	(* 12722 *)
	wTafterAlkaliWater  			AT %MW436:		WORD;	(* 12724 *)
	wConcAfterAlkaliWaterSet  	AT %MW438:		REAL;	(* 12726 *)
	wTsteril 						AT %MW440:		WORD;	(* 12728 *)
	wFlawSteril 					AT %MW442:		REAL;	(* 12730 *)
	wSterilTime 					AT %MW446:		WORD;	(* 12734 *)
	wDissolLineAccid 			AT %MW448:		WORD;	(* 12736 *)
	wDissolLineAlkali 			AT %MW450:		WORD;	(* 12738 *)
	xDissilDoAccid 				AT %MW452:		BOOL;		(* 12740 *)
	xDissolDoAlkali 				AT %MW454:		BOOL;		(* 12742 *)
	rConcSteril 					AT %MW444:		REAL;		(* 12732 *)
	rFlawWaterAfterAlcaliSet		AT %MW456	:	REAL;	(*	12744	*)
	rFlawWaterAfterAccidSet		AT %MW458	:	REAL;	(*	12746	*)
	rWaterAfterSterilFlaw			AT %MW460	:	REAL;	(*	12748	*)
	rWaterAfterSterilConc			AT %MW462	:	REAL;	(*	12750	*)
	rWaterAfterSterilT				AT %MW464	:	WORD;	(*	12752	*)
	rWaterAfterSterilTime			AT %MW466	:	WORD;	(*	12754	*)
	wConcPumpTimeSteril		AT %MW468	:	WORD;	(*	12756	*)







END_VAR

(* Global variable list: HMI_Sensors *)
VAR_GLOBAL

	Conc_Line1	AT %MW1100	:	REAL;	(*	13388	*)
	Conc_Line2	AT %MW1102	:	REAL;	(*	13390	*)
	Conc_Line3	AT %MW1104	:	REAL;	(*	13392	*)
	Conc_Line4	AT %MW1106	:	REAL;	(*	13394	*)

	CleanWaterLevel		AT %MW1108	:	REAL;	(*	13396	*)
	UsedWaterLevel		AT %MW1110	:	REAL;	(*	13398	*)
	AccidLevel		AT %MW1112	:	REAL;	(*	13400	*)
	AlkaliLevel		AT %MW1114	:	REAL;	(*	13402	*)

	Temp_Accid	AT %MW1116	:	REAL;	(*	13404	*)
	Temp_Alkali	AT %MW1118	:	REAL;	(*	13406	*)
	Temp_Line3	AT %MW1120	:	REAL;	(*	13408	*)
	Temp_Line4	AT %MW1122	:	REAL;	(*	13410	*)

	DI_FeedBackSwitchLine1	AT %MW1124	:	BOOL;	(*	13412	*)
	DI_FeedBackSwitchLine2	AT %MW1126	:	BOOL;	(*	13414	*)
	DI_FeedBackSwitchLine3	AT %MW1128	:	BOOL;	(*	13416	*)
	DI_FeedBackSwitchLine4	AT %MW1130	:	BOOL;	(*	13418	*)

	DI_AlkaliUpperLevel		AT %MW1132	:	BOOL;	(*	13420	*)
	DI_AccidUpperLevel		AT %MW1134	:	BOOL;	(*	13422	*)
	DI_WaterUpperLevel		AT %MW1136	:	BOOL;	(*	13424	*)
	DI_UsedWaterUpperLevel		AT %MW1138	:	BOOL;	(*	13426	*)



END_VAR

(* Global variable list: HMI_Settings *)
VAR_GLOBAL
END_VAR
VAR_GLOBAL RETAIN

	rDissolAlkaliConcSet 					AT %MW500:		REAL;	(* 12788 *)
	rDissolWaterConcSet 				AT %MW502:		REAL;	(* 12790 *)
	rDissolAccidConcSet 					AT %MW504:		REAL;	(* 12792 *)

	rDissolAccidLevelSet 					AT %MW562	:	REAL;	(*	12850	*)
	rDissolAlkaliLevelSet 					AT %MW564	:	REAL;	(*	12852	*)
	rPA_WorkTime_Acc					AT %MW566	:	WORD;	(*	12854	*)
	rPA_WorkTime_Alk					AT %MW568	:	WORD;	(*	12856	*)
	rConcCheckTime						AT %MW570	:	WORD;	(*	12858	*)


	wFlawSelWafing 						AT %MW506:		REAL;	(* 12794 *)
	wFlawDissolving 						AT %MW508:		REAL;	(* 12796 *)
	wUsedWaterLevelOK  				AT %MW510:		REAL:=90;	(* 12798 *)
	wUsedWaterLevelNotOK  			AT %MW512:		REAL:=80;	(* 12800 *)
	wAfterRinseConcAlk  					AT %MW514:		REAL:=30;	(* 12802 *)
	wAfterRinseConcAcc  				AT %MW516:		REAL:=30;	(* 12804 *)

	Heater_Kp								AT %MW518:		REAL:=5;	(* 12806 *)
	Heater_Ki								AT %MW520:		REAL:=3;	(* 12808 *)
	Heater_Kd								AT %MW522:		REAL;	(* 12810 *)
	Heater_wMaxPower 					AT %MW524:		WORD:=100;	(* 12812 *)
	Heater_wMinPower 					AT %MW526:		WORD;	(* 12814 *)
	Pump_Kp								AT %MW528:		REAL:=0.1;	(* 12816 *)
	Pump_Ki								AT %MW530:		REAL:=15;	(* 12818 *)
	Pump_Kd								AT %MW532:		REAL;	(* 12820 *)
	Pump_MaxSpeed 					AT %MW534:		WORD:=45;	(* 12822 *)
	Pump_MinSpeed 						AT %MW536:		WORD;	(* 12824 *)

	RemotePumpOnDelay				AT %MW572	:	WORD;	(*	12860	*)
	RemotePumpOffDelay				AT %MW574	:	WORD;	(*	12862	*)

	RemotePumpOnDelay2				AT %MW1572	:	WORD;	(*	12860	*)
	RemotePumpOffDelay2				AT %MW1574	:	WORD;	(*	12862	*)
	rConcSolutionStartOperationAlk		AT %MW576	:	REAL:=0.5;	(*	12864	*)
	rConcSolutionStopoperationAlk		AT %MW578	:	REAL:=0.5;	(*	12866	*)
	rConcSolutionStartOperationAcc		AT %MW580	:	REAL:=0.5;	(*	12868	*)
	rConcSolutionStopoperationAcc		AT %MW582	:	REAL:=0.5;	(*	12870	*)







	SelfWashUsedWaterLevelOK 		AT %MW538:		REAL;	(* 12826 *)
	SelfWashWaterLevelOK 				AT %MW540:		REAL;	(* 12828 *)
	SelfWashUsedWaterLevelDrain 		AT %MW542:		REAL:=0.01;	(* 12830 *)
	SelfWashWaterLevelDrain 			AT %MW544:		REAL:=0.01;	(* 12832 *)
	SelfWashAlkaliLevelOK 				AT %MW546:		REAL;	(* 12834 *)
	SelfWashAlkaliLevelDrain 			AT %MW548:		REAL;	(* 12836 *)
	SelfWashAccidLevelOK 				AT %MW550:		REAL;	(* 12838 *)
	SelfWashwAccidLevelDrain 			AT %MW552:		REAL;	(* 12840 *)
	SelfWashwPumpFlawSet 			AT %MW554:		REAL;	(* 12842 *)
	SelfWashByAlkaliTime  				AT %MW1556:		WORD;	(* 13844 *)
	SelfWashByAccidTime  				AT %MW1558:		WORD;	(* 13846 *)
	SelfWashByWaterTime_  				AT %MW1560:		WORD;	(* 13848 *)
	rWaterLevelNotOK 					AT %MW1562:		REAL:=90;	(* 12850 *)
	_SelfWashByWaterTime				AT %MW1200:		WORD;	(* 13848 *)

END_VAR

(* Global variable list: HMI_Values *)
VAR_GLOBAL

	xAlkaliIsReady:			BOOL;
	xAccidIsReady:			BOOL;

	xDrainOk:					BOOL;
	wDaysRemain:			WORD;
END_VAR

(* Global variable list: HMI_Valves *)
VAR_GLOBAL

	OnManual_V101	AT %MW700	:	BOOL;	(*	12988	*)
	OnManual_V102	AT %MW701	:	BOOL;	(*	12989	*)
	OnManual_V103	AT %MW702	:	BOOL;	(*	12990	*)
	OnManual_V104	AT %MW703	:	BOOL;	(*	12991	*)
	OnManual_V105	AT %MW704	:	BOOL;	(*	12992	*)
	OnManual_V106	AT %MW705	:	BOOL;	(*	12993	*)
	OnManual_V107	AT %MW706	:	BOOL;	(*	12994	*)
	OnManual_V108	AT %MW707	:	BOOL;	(*	12995	*)
	OnManual_V109	AT %MW708	:	BOOL;	(*	12996	*)
	OnManual_V110	AT %MW709	:	BOOL;	(*	12997	*)
	OnManual_V111	AT %MW710	:	BOOL;	(*	12998	*)
	OnManual_V201	AT %MW711	:	BOOL;	(*	12999	*)
	OnManual_V202	AT %MW712	:	BOOL;	(*	13000	*)
	OnManual_V203	AT %MW713	:	BOOL;	(*	13001	*)
	OnManual_V204	AT %MW714	:	BOOL;	(*	13002	*)
	OnManual_V205	AT %MW715	:	BOOL;	(*	13003	*)
	OnManual_V206	AT %MW716	:	BOOL;	(*	13004	*)
	OnManual_V207	AT %MW717	:	BOOL;	(*	13005	*)
	OnManual_V208	AT %MW718	:	BOOL;	(*	13006	*)
	OnManual_V209	AT %MW719	:	BOOL;	(*	13007	*)
	OnManual_V210	AT %MW720	:	BOOL;	(*	13008	*)
	OnManual_V211	AT %MW721	:	BOOL;	(*	13009	*)
	OnManual_V301	AT %MW722	:	BOOL;	(*	13010	*)
	OnManual_V302	AT %MW723	:	BOOL;	(*	13011	*)
	OnManual_V303	AT %MW724	:	BOOL;	(*	13012	*)
	OnManual_V304	AT %MW725	:	BOOL;	(*	13013	*)
	OnManual_V305	AT %MW726	:	BOOL;	(*	13014	*)
	OnManual_V306	AT %MW727	:	BOOL;	(*	13015	*)
	OnManual_V307	AT %MW728	:	BOOL;	(*	13016	*)
	OnManual_V308	AT %MW729	:	BOOL;	(*	13017	*)
	OnManual_V309	AT %MW730	:	BOOL;	(*	13018	*)
	OnManual_V310	AT %MW731	:	BOOL;	(*	13019	*)
	OnManual_V311	AT %MW732	:	BOOL;	(*	13020	*)
	OnManual_V401	AT %MW733	:	BOOL;	(*	13021	*)
	OnManual_V402	AT %MW734	:	BOOL;	(*	13022	*)
	OnManual_V403	AT %MW735	:	BOOL;	(*	13023	*)
	OnManual_V404	AT %MW736	:	BOOL;	(*	13024	*)
	OnManual_V405	AT %MW737	:	BOOL;	(*	13025	*)
	OnManual_V406	AT %MW738	:	BOOL;	(*	13026	*)
	OnManual_V407	AT %MW739	:	BOOL;	(*	13027	*)
	OnManual_V408	AT %MW740	:	BOOL;	(*	13028	*)
	OnManual_V409	AT %MW741	:	BOOL;	(*	13029	*)
	OnManual_V410	AT %MW742	:	BOOL;	(*	13030	*)
	OnManual_V411	AT %MW743	:	BOOL;	(*	13031	*)
	OnManual_V501	AT %MW744	:	BOOL;	(*	13032	*)
	OnManual_V510	AT %MW745	:	BOOL;	(*	13033	*)
	OnManual_V511	AT %MW746	:	BOOL;	(*	13034	*)
	OnManual_V512	AT %MW747	:	BOOL;	(*	13035	*)
	OnManual_V513	AT %MW748	:	BOOL;	(*	13036	*)
	OnManual_V514	AT %MW749	:	BOOL;	(*	13037	*)
	OnManual_V515	AT %MW750	:	BOOL;	(*	13038	*)
							
							
							
							
	xState_V101	AT %MW751	:	BOOL;	(*	13039	*)
	xState_V102	AT %MW752	:	BOOL;	(*	13040	*)
	xState_V103	AT %MW753	:	BOOL;	(*	13041	*)
	xState_V104	AT %MW754	:	BOOL;	(*	13042	*)
	xState_V105	AT %MW755	:	BOOL;	(*	13043	*)
	xState_V106	AT %MW756	:	BOOL;	(*	13044	*)
	xState_V107	AT %MW757	:	BOOL;	(*	13045	*)
	xState_V108	AT %MW758	:	BOOL;	(*	13046	*)
	xState_V109	AT %MW759	:	BOOL;	(*	13047	*)
	xState_V110	AT %MW760	:	BOOL;	(*	13048	*)
	xState_V111	AT %MW761	:	BOOL;	(*	13049	*)
	xState_V201	AT %MW762	:	BOOL;	(*	13050	*)
	xState_V202	AT %MW763	:	BOOL;	(*	13051	*)
	xState_V203	AT %MW764	:	BOOL;	(*	13052	*)
	xState_V204	AT %MW765	:	BOOL;	(*	13053	*)
	xState_V205	AT %MW766	:	BOOL;	(*	13054	*)
	xState_V206	AT %MW767	:	BOOL;	(*	13055	*)
	xState_V207	AT %MW768	:	BOOL;	(*	13056	*)
	xState_V208	AT %MW769	:	BOOL;	(*	13057	*)
	xState_V209	AT %MW770	:	BOOL;	(*	13058	*)
	xState_V210	AT %MW771	:	BOOL;	(*	13059	*)
	xState_V211	AT %MW772	:	BOOL;	(*	13060	*)
	xState_V301	AT %MW773	:	BOOL;	(*	13061	*)
	xState_V302	AT %MW774	:	BOOL;	(*	13062	*)
	xState_V303	AT %MW775	:	BOOL;	(*	13063	*)
	xState_V304	AT %MW776	:	BOOL;	(*	13064	*)
	xState_V305	AT %MW777	:	BOOL;	(*	13065	*)
	xState_V306	AT %MW778	:	BOOL;	(*	13066	*)
	xState_V307	AT %MW779	:	BOOL;	(*	13067	*)
	xState_V308	AT %MW780	:	BOOL;	(*	13068	*)
	xState_V309	AT %MW781	:	BOOL;	(*	13069	*)
	xState_V310	AT %MW782	:	BOOL;	(*	13070	*)
	xState_V311	AT %MW783	:	BOOL;	(*	13071	*)
	xState_V401	AT %MW784	:	BOOL;	(*	13072	*)
	xState_V402	AT %MW785	:	BOOL;	(*	13073	*)
	xState_V403	AT %MW786	:	BOOL;	(*	13074	*)
	xState_V404	AT %MW787	:	BOOL;	(*	13075	*)
	xState_V405	AT %MW788	:	BOOL;	(*	13076	*)
	xState_V406	AT %MW789	:	BOOL;	(*	13077	*)
	xState_V407	AT %MW790	:	BOOL;	(*	13078	*)
	xState_V408	AT %MW791	:	BOOL;	(*	13079	*)
	xState_V409	AT %MW792	:	BOOL;	(*	13080	*)
	xState_V410	AT %MW793	:	BOOL;	(*	13081	*)
	xState_V411	AT %MW794	:	BOOL;	(*	13082	*)
	xState_V501	AT %MW795	:	BOOL;	(*	13083	*)
	xState_V510	AT %MW796	:	BOOL;	(*	13084	*)
	xState_V511	AT %MW797	:	BOOL;	(*	13085	*)
	xState_V512	AT %MW798	:	BOOL;	(*	13086	*)
	xState_V513	AT %MW799	:	BOOL;	(*	13087	*)
	xState_V514	AT %MW800	:	BOOL;	(*	13088	*)
	xState_V515	AT %MW801	:	BOOL;	(*	13089	*)
							
							
	OnAuto_V101	AT %MW802	:	BOOL;	(*	13090	*)
	OnAuto_V102	AT %MW803	:	BOOL;	(*	13091	*)
	OnAuto_V103	AT %MW804	:	BOOL;	(*	13092	*)
	OnAuto_V104	AT %MW805	:	BOOL;	(*	13093	*)
	OnAuto_V105	AT %MW806	:	BOOL;	(*	13094	*)
	OnAuto_V106	AT %MW807	:	BOOL;	(*	13095	*)
	OnAuto_V107	AT %MW808	:	BOOL;	(*	13096	*)
	OnAuto_V108	AT %MW809	:	BOOL;	(*	13097	*)
	OnAuto_V109	AT %MW810	:	BOOL;	(*	13098	*)
	OnAuto_V110	AT %MW811	:	BOOL;	(*	13099	*)
	OnAuto_V111	AT %MW812	:	BOOL;	(*	13100	*)
	OnAuto_V201	AT %MW813	:	BOOL;	(*	13101	*)
	OnAuto_V202	AT %MW814	:	BOOL;	(*	13102	*)
	OnAuto_V203	AT %MW815	:	BOOL;	(*	13103	*)
	OnAuto_V204	AT %MW816	:	BOOL;	(*	13104	*)
	OnAuto_V205	AT %MW817	:	BOOL;	(*	13105	*)
	OnAuto_V206	AT %MW818	:	BOOL;	(*	13106	*)
	OnAuto_V207	AT %MW819	:	BOOL;	(*	13107	*)
	OnAuto_V208	AT %MW820	:	BOOL;	(*	13108	*)
	OnAuto_V209	AT %MW821	:	BOOL;	(*	13109	*)
	OnAuto_V210	AT %MW822	:	BOOL;	(*	13110	*)
	OnAuto_V211	AT %MW823	:	BOOL;	(*	13111	*)
	OnAuto_V301	AT %MW824	:	BOOL;	(*	13112	*)
	OnAuto_V302	AT %MW825	:	BOOL;	(*	13113	*)
	OnAuto_V303	AT %MW826	:	BOOL;	(*	13114	*)
	OnAuto_V304	AT %MW827	:	BOOL;	(*	13115	*)
	OnAuto_V305	AT %MW828	:	BOOL;	(*	13116	*)
	OnAuto_V306	AT %MW829	:	BOOL;	(*	13117	*)
	OnAuto_V307	AT %MW830	:	BOOL;	(*	13118	*)
	OnAuto_V308	AT %MW831	:	BOOL;	(*	13119	*)
	OnAuto_V309	AT %MW832	:	BOOL;	(*	13120	*)
	OnAuto_V310	AT %MW833	:	BOOL;	(*	13121	*)
	OnAuto_V311	AT %MW834	:	BOOL;	(*	13122	*)
	OnAuto_V401	AT %MW835	:	BOOL;	(*	13123	*)
	OnAuto_V402	AT %MW836	:	BOOL;	(*	13124	*)
	OnAuto_V403	AT %MW837	:	BOOL;	(*	13125	*)
	OnAuto_V404	AT %MW838	:	BOOL;	(*	13126	*)
	OnAuto_V405	AT %MW839	:	BOOL;	(*	13127	*)
	OnAuto_V406	AT %MW840	:	BOOL;	(*	13128	*)
	OnAuto_V407	AT %MW841	:	BOOL;	(*	13129	*)
	OnAuto_V408	AT %MW842	:	BOOL;	(*	13130	*)
	OnAuto_V409	AT %MW843	:	BOOL;	(*	13131	*)
	OnAuto_V410	AT %MW844	:	BOOL;	(*	13132	*)
	OnAuto_V411	AT %MW845	:	BOOL;	(*	13133	*)
	OnAuto_V501	AT %MW846	:	BOOL;	(*	13134	*)
	OnAuto_V510	AT %MW847	:	BOOL;	(*	13135	*)
	OnAuto_V511	AT %MW848	:	BOOL;	(*	13136	*)
	OnAuto_V512	AT %MW849	:	BOOL;	(*	13137	*)
	OnAuto_V513	AT %MW850	:	BOOL;	(*	13138	*)
	OnAuto_V514	AT %MW851	:	BOOL;	(*	13139	*)
	OnAuto_V515	AT %MW852	:	BOOL;	(*	13140	*)



	xStopFillingWaterTank: BOOL;



END_VAR

VAR_GLOBAL RETAIN PERSISTENT

	ManualMode_V101	AT %MW853	:	BOOL;	(*	13140	*)
	ManualMode_V102	AT %MW854	:	BOOL;	(*	13141	*)
	ManualMode_V103	AT %MW855	:	BOOL;	(*	13142	*)
	ManualMode_V104	AT %MW856	:	BOOL;	(*	13143	*)
	ManualMode_V105	AT %MW857	:	BOOL;	(*	13144	*)
	ManualMode_V106	AT %MW858	:	BOOL;	(*	13145	*)
	ManualMode_V107	AT %MW859	:	BOOL;	(*	13146	*)
	ManualMode_V108	AT %MW860	:	BOOL;	(*	13147	*)
	ManualMode_V109	AT %MW861	:	BOOL;	(*	13148	*)
	ManualMode_V110	AT %MW862	:	BOOL;	(*	13149	*)
	ManualMode_V111	AT %MW863	:	BOOL;	(*	13150	*)
	ManualMode_V201	AT %MW864	:	BOOL;	(*	13151	*)
	ManualMode_V202	AT %MW865	:	BOOL;	(*	13152	*)
	ManualMode_V203	AT %MW866	:	BOOL;	(*	13153	*)
	ManualMode_V204	AT %MW867	:	BOOL;	(*	13154	*)
	ManualMode_V205	AT %MW868	:	BOOL;	(*	13155	*)
	ManualMode_V206	AT %MW869	:	BOOL;	(*	13156	*)
	ManualMode_V207	AT %MW870	:	BOOL;	(*	13157	*)
	ManualMode_V208	AT %MW871	:	BOOL;	(*	13158	*)
	ManualMode_V209	AT %MW872	:	BOOL;	(*	13159	*)
	ManualMode_V210	AT %MW873	:	BOOL;	(*	13160	*)
	ManualMode_V211	AT %MW874	:	BOOL;	(*	13161	*)
	ManualMode_V301	AT %MW875	:	BOOL;	(*	13162	*)
	ManualMode_V302	AT %MW876	:	BOOL;	(*	13163	*)
	ManualMode_V303	AT %MW877	:	BOOL;	(*	13164	*)
	ManualMode_V304	AT %MW878	:	BOOL;	(*	13165	*)
	ManualMode_V305	AT %MW879	:	BOOL;	(*	13166	*)
	ManualMode_V306	AT %MW880	:	BOOL;	(*	13167	*)
	ManualMode_V307	AT %MW881	:	BOOL;	(*	13168	*)
	ManualMode_V308	AT %MW882	:	BOOL;	(*	13169	*)
	ManualMode_V309	AT %MW883	:	BOOL;	(*	13170	*)
	ManualMode_V310	AT %MW884	:	BOOL;	(*	13171	*)
	ManualMode_V311	AT %MW885	:	BOOL;	(*	13172	*)
	ManualMode_V401	AT %MW886	:	BOOL;	(*	13173	*)
	ManualMode_V402	AT %MW887	:	BOOL;	(*	13174	*)
	ManualMode_V403	AT %MW888	:	BOOL;	(*	13175	*)
	ManualMode_V404	AT %MW889	:	BOOL;	(*	13176	*)
	ManualMode_V405	AT %MW890	:	BOOL;	(*	13177	*)
	ManualMode_V406	AT %MW891	:	BOOL;	(*	13178	*)
	ManualMode_V407	AT %MW892	:	BOOL;	(*	13179	*)
	ManualMode_V408	AT %MW893	:	BOOL;	(*	13180	*)
	ManualMode_V409	AT %MW894	:	BOOL;	(*	13181	*)
	ManualMode_V410	AT %MW895	:	BOOL;	(*	13182	*)
	ManualMode_V411	AT %MW896	:	BOOL;	(*	13183	*)
	ManualMode_V501	AT %MW897	:	BOOL;	(*	13184	*)
	ManualMode_V510	AT %MW898	:	BOOL;	(*	13185	*)
	ManualMode_V511	AT %MW899	:	BOOL;	(*	13186	*)
	ManualMode_V512	AT %MW900	:	BOOL;	(*	13187	*)
	ManualMode_V513	AT %MW901	:	BOOL;	(*	13188	*)
	ManualMode_V514	AT %MW902	:	BOOL;	(*	13189	*)
	ManualMode_V515	AT %MW903	:	BOOL;	(*	13190	*)


END_VAR

(* Global variable list: ProcGlobal *)
VAR_GLOBAL
	xDissolving_StartLine1:		BOOL;
	xDissolving_StartLine2:		BOOL;
	xDissolving_StartLine3:		BOOL;
	xDissolving_StartLine4:		BOOL;

	xDissolving_PausetLine1:		BOOL;
	xDissolving_PausetLine2:		BOOL;
	xDissolving_PausetLine3:		BOOL;
	xDissolving_PausetLine4:		BOOL;


	xDoAccid_Line1:					BOOL;
	xDoAlkali_Line1:					BOOL;
	xDoAccid_Line2:					BOOL;
	xDoAlkali_Line2:					BOOL;
	xDoAccid_Line3:					BOOL;
	xDoAlkali_Line3:					BOOL;
	xDoAccid_Line4:					BOOL;
	xDoAlkali_Line4:					BOOL;





END_VAR
VAR_GLOBAL RETAIN
	xAccidIsGoing1:					BOOL;
	xAccidIsGoing2:					BOOL;
	xAccidIsGoing3:					BOOL;
	xAccidIsGoing4:					BOOL;
END_VAR

(* Global variable list: Pump *)
VAR_GLOBAL

	Pump_FlawAutoSet_1:		REAL;
	Pump_FlawAutoSet_2:		REAL;
	Pump_FlawAutoSet_3:		REAL;
	Pump_FlawAutoSet_4:		REAL;



END_VAR

(* Global variable list: RecipeVars *)
VAR_GLOBAL

	arOperations:					ARRAY[0..7] OF BOOL;




END_VAR

VAR_GLOBAL RETAIN

	arAlkaliTime:					ARRAY[1..4, 1..10] OF WORD;
	arTalkaliSet: 					ARRAY[1..4, 1..10] OF WORD;
	arFlawAlkaliSet: 				ARRAY[1..4, 1..10] OF REAL;
	arConcAlkaliSet: 				ARRAY[1..4, 1..10] OF REAL;

	arAccidTime:					ARRAY[1..4, 1..10] OF WORD;
	arTaccidSet: 					ARRAY[1..4, 1..10] OF WORD;
	arFlawAccidSet: 				ARRAY[1..4, 1..10] OF REAL;
	arConcAccidSet:				ARRAY[1..4, 1..10] OF REAL;

	arWaterTime: 					ARRAY[1..4, 1..10] OF WORD;
	arTwaterSet: 					ARRAY[1..4, 1..10] OF WORD;
	arFlawWaterSet: 				ARRAY[1..4, 1..10] OF REAL;

	arAfterAccidWaterTime: 		ARRAY[1..4, 1..10] OF WORD;
	arTafterAccidWater: 			ARRAY[1..4, 1..10] OF WORD;
	arConcAfterAccidWaterSet: 	ARRAY[1..4, 1..10] OF REAL;

	arAfterAlkaliWaterTime: 		ARRAY[1..4, 1..10] OF WORD;
	arTafterAlkaliWater: 			ARRAY[1..4, 1..10] OF WORD;
	arConcAfterAlkaliWaterSet: 	ARRAY[1..4, 1..10] OF REAL;

	arTsterilSet: 					ARRAY[1..4, 1..10] OF WORD;
	arFlawSterilSet: 				ARRAY[1..4, 1..10] OF REAL;
	arConcSterilSet: 				ARRAY[1..4, 1..10] OF REAL;
	arSterilTime: 					ARRAY[1..4, 1..10] OF WORD;

	arFlawWaterAfterAlcaliSet:	ARRAY[1..4, 1..10] OF REAL;
	arFlawWaterAfterAccidSet:	ARRAY[1..4, 1..10] OF REAL;

	arWaterAfterSterilFlaw:		ARRAY[1..4, 1..10] OF REAL;
	arWaterAfterSterilConc:		ARRAY[1..4, 1..10] OF REAL;
	arWaterAfterSterilT:			ARRAY[1..4, 1..10] OF WORD;
	arWaterAfterSterilTime:		ARRAY[1..4, 1..10] OF WORD;
	arConcPumpTimeSteril:		ARRAY[1..4, 1..10] OF WORD;
	arOperations2x:				ARRAY[1..4,0..7] OF BOOL;
	arOperations3x:				ARRAY[1..4,1..10,0..7] OF BOOL;


END_VAR

(* Data type *)
TYPE Dissolving_States :
(
	DissolvingStop:=0,
	WaterStart:=1,
	AlkaliTankFullUp:=2,
	AlkaliConc:=3,
	AlkaliConcMessure:=4,
	WaterAfter:=5,
	AccidTankFullUp:=6,
	AccidConc:=7,
	AccidConcMessure:=8,
	DissolvingPause:=9
);
END_TYPE

(* Data type *)
TYPE SelfWashingStates :
(
	StopSelfWashing:=0,
	FillUsedWaterTank:=1,
	FillWaterTank:=2,
	FillAccidTank:=3,
	FillAlkaliTank:=4,
	WashUsedWaterTankAlkali:=5,
	WashUsedWaterTankAccid:=6,
	WashUsedWaterTankWater:=7,
	WashWaterTankAlkali:=8,
	WashWaterTankAccid:=9,
	WashWaterTankWater:=10,
	WashAlkaliTankAccid:=11,
	WashAlkaliTankWater:=12,
	WashAccidTankAlkali:=13,
	WashAccidTankWater:=14,
	CheckAlkali:=15,
	CheckAccid:=16,
	CheckAll:=17,
	WaitAlkaliDissolving:=18,
	WaitAccidDissolving:=19,
	WaitAllDissolving:=20,
	EmptyUsedWaterTank:=21,
	EmptyWaterTank:=22,
	EmptyAlkaliTank:=23,
	EmptyAccidTank:=24,
	WaitManualAlkaliDrain:=25,
	WaitManualAccidDrain:=26,
	WaterFinalDrain:=27,
	UsedWaterFinalDrain:=28,
	AlkaliFinalDrain:=29,
	AccidFinalDrain:=30,
	WaitManualAlkaliDrainFinal:=31,
	WaitManualAccidDrainFinal:=32,
	SelfWashingPause:=33
);
END_TYPE

(* Data type *)
TYPE WashingProcess_States :
(
	Washing_Stop				:= 0,	(* неопределенном состоянии, не выполняется *)
	Rinse 		:= 1,	(*ожидание остаточного давления *)

	AlkaliIn			:= 2, 	(*установка и прокачка газа*)
	WaterAfterAlkalin	:= 3,	(*включение коммутатора	*)
	Accid	:= 4, 	(*включение блока питания магнетрона	*)
	WaterAfterAccid		:= 5,	(*напыление магнетроном*)
	Sterelisation:= 6,
	WaterAfterSterilisation:=7,

	RinseUsedWater	:= 8,	(*включение блока питания компенсатора *)
	AlkaliInPushing:=9,
	AlkaliInWashing:=10,
	AccidPushing:=11,
	AccidWashing:=12,
	HotWaterSterilisation:=13,
	SolutionSterilisation:=14,
	FindNextOperation	:= 15,	(*включение блока питания ассистента	*)
	WashingPause:=16,
	CheckWaterLevel:=17
);
END_TYPE

(* POU PLC_PRG, ST *)
PROGRAM PLC_PRG
VAR
	dDate:	DT;
	dDateStop:DT:=DT#2020-02-16-08:00:00;
	CurTimeEx_:CurTimeEx;
	SystemTimeDate_:SystemTimeDate;
	SysTime64_:SysTime64;
	xOutOff:	BOOL;
END_VAR
InToVars();

prDevice();
prProcess();
prValue_to_AO();


dDate:=SysRtcGetTime(TRUE);

IF dDateStop > dDate THEN
	xOutOff:=TRUE;
END_IF
(*
CurTimeEx_(SystemTime:=SysTime64_ , TimeDate:= SystemTimeDate_);
IF SystemTimeDate_.Month = 2 THEN
	wDaysRemain:= 27 - SystemTimeDate_.Day(* + 16*);
	IF SystemTimeDate_.Day > 27 THEN
		wDaysRemain:=0;
	END_IF
ELSIF SystemTimeDate_.Month = 3 THEN
	(*wDaysRemain:=16 - SystemTimeDate_.Day;
	IF SystemTimeDate_.Day > 16 THEN
		wDaysRemain:=0;
	END_IF*)
	wDaysRemain:=0;
ELSE
	wDaysRemain:=0;
END_IF

Simulation();


IF wDaysRemain > 0 THEN
	VarsToOut();
END_IF
*)

VarsToOut();


xResetAlmAll:=FALSE;
END_PROGRAM

(* POU InToVars, ST *)
PROGRAM InToVars
VAR

END_VAR
DI_AlkaliUpperLevel:= NOT _LH_2;
DI_AccidUpperLevel:= NOT _LH_1;



DI_FeedBackSwitchLine1:= _DI_FeedBackSwitchLine1;
DI_FeedBackSwitchLine2:= _DI_FeedBackSwitchLine2;
DI_FeedBackSwitchLine3:= _DI_FeedBackSwitchLine3;
DI_FeedBackSwitchLine4:= _DI_FeedBackSwitchLine4;


DI_WaterUpperLevel:= NOT _LH_3;
DI_UsedWaterUpperLevel:= NOT _LH_4;


DI_V101:= NOT _DI_V101;
DI_V102:= NOT _DI_V102;
DI_V103:= NOT _DI_V103;
DI_V104:= NOT _DI_V104;
DI_V105:= NOT _DI_V105;
DI_V106:= NOT _DI_V106;
DI_V107:= NOT _DI_V107;
DI_V108:= NOT _DI_V108;
DI_V109:= NOT _DI_V109;
DI_V110:= NOT _DI_V110;
DI_V111:= NOT _DI_V111;
DI_V201:= NOT _DI_V201;
DI_V202:= NOT _DI_V202;
DI_V203:= NOT _DI_V203;
DI_V204:= NOT _DI_V204;
DI_V205:= NOT _DI_V205;
DI_V206:= NOT _DI_V206;
DI_V207:= NOT _DI_V207;
DI_V208:= NOT _DI_V208;
DI_V209:= NOT _DI_V209;
DI_V210:= NOT _DI_V210;
DI_V211:= NOT _DI_V211;
DI_V301:= NOT _DI_V301;
DI_V302:= NOT _DI_V302;
DI_V303:= NOT _DI_V303;
DI_V304:= NOT _DI_V304;
DI_V305:= NOT _DI_V305;
DI_V306:= NOT _DI_V306;
DI_V307:= NOT _DI_V307;
DI_V308:= NOT _DI_V308;
DI_V309:= NOT _DI_V309;
DI_V310:= NOT _DI_V310;
DI_V311:= NOT _DI_V311;
DI_V401:= NOT _DI_V401;
DI_V402:= NOT _DI_V402;
DI_V403:= NOT _DI_V403;
DI_V404:= NOT _DI_V404;
DI_V405:= NOT _DI_V405;
DI_V406:= NOT _DI_V406;
DI_V407:= NOT _DI_V407;
DI_V408:= NOT _DI_V408;
DI_V409:= NOT _DI_V409;
DI_V410:= NOT _DI_V410;
DI_V411:= NOT _DI_V411;
DI_V501:= NOT _DI_V501;
DI_V510:= NOT _DI_V510;
DI_V511:= NOT _DI_V511;
DI_V512:= NOT _DI_V512;
DI_V513:= NOT _DI_V513;
DI_V514:= NOT _DI_V514;
DI_V515:= NOT _DI_V515;


Pump_InvNorm_1:= _Pump_Alm_1;
Pump_InvNorm_2:= _Pump_Alm_2;
Pump_InvNorm_3:= _Pump_Alm_3;
Pump_InvNorm_4:= _Pump_Alm_4;


Pump_FeedbackOn_1:=_Pump_FeedbackOn_1;
Pump_FeedbackOn_2:=_Pump_FeedbackOn_2;
Pump_FeedbackOn_3:=_Pump_FeedbackOn_3;
Pump_FeedbackOn_4:=_Pump_FeedbackOn_4;


AI_Conc_Line1:= _AI_Conc_Line1;
AI_Conc_Line2:= _AI_Conc_Line2;
AI_Conc_Line3:= _AI_Conc_Line3;
AI_Conc_Line4:= _AI_Conc_Line4;

AI_CleanWaterLevel:= _AI_CleanWaterLevel;
AI_UsedWaterLevel:= _AI_UsedWaterLevel;
AI_AccidLevel:= _AI_AccidLevel;
AI_AlkaliLevel:= _AI_AlkaliLevel;






AI_Temp_Accid:= _AI_Temp_Accid;
AI_Temp_Alkali:= _AI_Temp_Alkali;
(*
AI_Temp_Line3:= _AI_Temp_Line3;
AI_Temp_Line4:= _AI_Temp_Line4;
*)

AI_Heater_Tget_1 := _AI_Heater_Tget_1 ;
AI_Heater_Tget_2 := _AI_Heater_Tget_2 ;
AI_Heater_Tget_3 := _AI_Heater_Tget_3 ;
AI_Heater_Tget_4 := _AI_Heater_Tget_4 ;
 
AI_Heater_BackTget_1:= _AI_Heater_BackTget_1;
AI_Heater_BackTget_2:= _AI_Heater_BackTget_2;
AI_Heater_BackTget_3:= _AI_Heater_BackTget_3;
AI_Heater_BackTget_4:= _AI_Heater_BackTget_4;
 
AI_Flaw_Line1:= _AI_Flaw_Line1;
AI_Flaw_Line2:= _AI_Flaw_Line2;
AI_Flaw_Line3:= _AI_Flaw_Line3;
AI_Flaw_Line4:= _AI_Flaw_Line4;

Permition_Line_1:=_Permition_Line_1;
Permition_Line_2:=_Permition_Line_2;
Permition_Line_3:=_Permition_Line_3;
Permition_Line_4:=_Permition_Line_4;
Permition_Line_5:=_Permition_Line_5;
END_PROGRAM

(* POU Device/prDevice, ST *)
PROGRAM prDevice
VAR
END_VAR
prSensors();
prHeater();

prPump();

prValve();
END_PROGRAM

(* POU Device/Sensors/prSensors, ST *)
PROGRAM prSensors
VAR
END_VAR
prFlaw();
prConc();
prLevel();
prTemperature();
END_PROGRAM

(* POU Device/Sensors/prFlaw, ST *)
PROGRAM prFlaw
VAR

	FlawMessure_1:	fb_sensor;
	FlawMessure_2:	fb_sensor;
	FlawMessure_3:	fb_sensor;
	FlawMessure_4:	fb_sensor;

	FlawMessure_Trafo_1: LIN_TRAFO;
	FlawMessure_Trafo_2: LIN_TRAFO;
	FlawMessure_Trafo_3: LIN_TRAFO;
	FlawMessure_Trafo_4: LIN_TRAFO;

END_VAR
(*
FlawMessure_1(
	remont:= , 
	use_pt100:= , 
	value:= AI_Flaw_Line1,
	value_20ma:= , 
	min_value:= ,
	max_value:=10 ,
	crash_value_4_20ma_1:= , 
	crash_value_4_20ma_2:= , 
	value_int:= , 
	crash_value_PT100_1:= , 
	crash_value_PT100_2:= , 
	sensor_offset:= , 
	sensor_gain:= , 
	rezult_value=> Pump_FlawGet_1,
	crash_value=> , 
	out_crash_int=> );

FlawMessure_2(
	remont:= ,
	use_pt100:= ,
	value:= AI_Flaw_Line2,
	value_20ma:= ,
	min_value:= ,
	max_value:=10 ,
	crash_value_4_20ma_1:= , 
	crash_value_4_20ma_2:= , 
	value_int:= , 
	crash_value_PT100_1:= , 
	crash_value_PT100_2:= , 
	sensor_offset:= , 
	sensor_gain:= , 
	rezult_value=> Pump_FlawGet_2,
	crash_value=> , 
	out_crash_int=> );

FlawMessure_3(
	remont:= , 
	use_pt100:= , 
	value:= AI_Flaw_Line3,
	value_20ma:= , 
	min_value:= ,
	max_value:=10 ,
	crash_value_4_20ma_1:= , 
	crash_value_4_20ma_2:= , 
	value_int:= , 
	crash_value_PT100_1:= , 
	crash_value_PT100_2:= , 
	sensor_offset:= , 
	sensor_gain:= , 
	rezult_value=> Pump_FlawGet_3,
	crash_value=> , 
	out_crash_int=> );

FlawMessure_4(
	remont:= , 
	use_pt100:= , 
	value:= AI_Flaw_Line4,
	value_20ma:= , 
	min_value:= ,
	max_value:=10 ,
	crash_value_4_20ma_1:= , 
	crash_value_4_20ma_2:= , 
	value_int:= , 
	crash_value_PT100_1:= , 
	crash_value_PT100_2:= , 
	sensor_offset:= , 
	sensor_gain:= , 
	rezult_value=> Pump_FlawGet_4,
	crash_value=> , 
	out_crash_int=> );
*)

FlawMessure_Trafo_1(
	IN:= AI_Flaw_Line1,
	IN_MIN:= 0,
	IN_MAX:= 32767,
	OUT_MIN:= 0,
	OUT_MAX:= 61 );
Pump_FlawGet_1:= FlawMessure_Trafo_1.OUT;
IF AI_Flaw_Line1 < 300 THEN
	Pump_FlawGet_1:=0;
END_IF


FlawMessure_Trafo_2(
	IN:= AI_Flaw_Line2,
	IN_MIN:= 0,
	IN_MAX:= 32767,
	OUT_MIN:= 0,
	OUT_MAX:= 61 );
Pump_FlawGet_2:= FlawMessure_Trafo_2.OUT;
IF AI_Flaw_Line2 < 300 THEN
	Pump_FlawGet_2:=0;
END_IF

FlawMessure_Trafo_3(
	IN:= AI_Flaw_Line3,
	IN_MIN:= 0,
	IN_MAX:= 32767,
	OUT_MIN:= 0,
	OUT_MAX:= 61 );
Pump_FlawGet_3:= FlawMessure_Trafo_3.OUT;
IF AI_Flaw_Line3 < 300 THEN
	Pump_FlawGet_3:=0;
END_IF

FlawMessure_Trafo_4(
	IN:= AI_Flaw_Line4,
	IN_MIN:= 0,
	IN_MAX:= 32767,
	OUT_MIN:= 0,
	OUT_MAX:= 61 );
Pump_FlawGet_4:= FlawMessure_Trafo_4.OUT;
IF AI_Flaw_Line4 < 300 THEN
	Pump_FlawGet_4:=0;
END_IF
END_PROGRAM

(* POU Device/Sensors/fb_sensor, ST *)
FUNCTION_BLOCK fb_sensor
VAR_INPUT

	remont	:						BOOL	;
	use_pt100	:					BOOL	;
	value	:						INT	;
	value_20ma	:				REAL	:=	32767.0	;
	min_value	:					REAL	;
	max_value	:					REAL	:=	100.0	;
	crash_value_4_20ma_1	:	INT	:=	32767	;
	crash_value_4_20ma_2	:	INT	:=	-32768	;
	value_int	:					INT	;
	crash_value_PT100_1	:	INT	:=	-2000	;
	crash_value_PT100_2	:	INT	:=	8500	;
	sensor_offset	:				REAL	;
	sensor_gain	:				REAL	:=	1.0	;
END_VAR
VAR_OUTPUT
	rezult_value	:				REAL	;
	crash_value	:				BOOL	;
	out_crash_int	:				WORD	;

END_VAR
VAR
	(*db_crash_to_int:				fb_crash_to_int;*)
END_VAR
(*fb для пересчета аналоговых датчиков*)
IF remont = FALSE
  THEN
    (*обрыв или кз датчика*)
    IF use_pt100 = FALSE
      THEN
        (*если датчик 4-20ма*)
        IF value = crash_value_4_20ma_1 OR value = crash_value_4_20ma_2
          THEN
            rezult_value:= 0;
            crash_value:=TRUE;
          ELSE
            rezult_value:= (min_value + INT_TO_REAL(value) * (max_value - min_value)/value_20ma) * sensor_gain + sensor_offset;
            crash_value:=FALSE;
        END_IF;
      ELSE
        (*если датчик РТ100*)
        IF value_int <=crash_value_PT100_1 OR value_int >= crash_value_PT100_2
          THEN
            rezult_value:= 0;
            crash_value:=TRUE;
          ELSE
            rezult_value:= sensor_offset + sensor_gain * (INT_TO_REAL(value_int)/10.0);
            crash_value:=FALSE;
        END_IF;
    END_IF;
  ELSE
    rezult_value:= 0;
    crash_value:=FALSE;
END_IF;

(*
(*аварии для панели*)
db_crash_to_int(
  crash_1:= crash_value );
out_crash_int:= db_crash_to_int.rezult_int_crash;
*)
END_FUNCTION_BLOCK

(* POU _ExtraFB/mathematical functions/LIN_TRAFO, ST *)
(* linear transformation *)
FUNCTION_BLOCK LIN_TRAFO
VAR_INPUT
	IN: REAL;				(* input value*)
	IN_MIN:REAL;			(* minimum input value *)
	IN_MAX:REAL;			(* maximum input value *)
	OUT_MIN:REAL;		(* corresponding minimum output value *)
	OUT_MAX:REAL;		(* corresponding maximum output value *)
END_VAR
VAR_OUTPUT
	OUT: REAL;			(* output value *)
	ERROR: BOOL;		(* error: IN_MIN = IN_MAX or IN out of interval *)
END_VAR

VAR
	Diff: REAL;
END_VAR
Diff := IN_MAX-IN_MIN;
ERROR := (Diff=0) OR (IN<IN_MIN) OR (IN>IN_MAX);

IF NOT ERROR THEN
	OUT := (IN-IN_MIN)/Diff * (OUT_MAX-OUT_MIN) + OUT_MIN;
END_IF
END_FUNCTION_BLOCK

(* POU Device/Sensors/prConc, ST *)
PROGRAM prConc
VAR

	Conc_Line_1: fb_sensor;
	Conc_Line_2: fb_sensor;
	Conc_Line_3: fb_sensor;
	Conc_Line_4: fb_sensor;

	ConcEnd_Line_1:	fb_concentrator;
	ConcEnd_Line_2:	fb_concentrator;
	ConcEnd_Line_3:	fb_concentrator;
	ConcEnd_Line_4:	fb_concentrator;

	Conc_Line1_raw: REAL;
	Conc_Line2_raw: REAL;
	Conc_Line3_raw: REAL;
	Conc_Line4_raw: REAL;

	AccidAlkaliSwitch_1: fbAccidAlkaliSwitch;
	AccidAlkaliSwitch_2: fbAccidAlkaliSwitch;
	AccidAlkaliSwitch_3: fbAccidAlkaliSwitch;
	AccidAlkaliSwitch_4: fbAccidAlkaliSwitch;

END_VAR
AccidAlkaliSwitch_1(
	xV_AccidOut:= xState_V103,
	xV_AlkaliOut:= xState_V104,
	xAccidOn:=xAccidIsGoing1 );

AccidAlkaliSwitch_2(
	xV_AccidOut:= xState_V203,
	xV_AlkaliOut:= xState_V204,
	xAccidOn:=xAccidIsGoing2 );

AccidAlkaliSwitch_3(
	xV_AccidOut:= xState_V303,
	xV_AlkaliOut:= xState_V304,
	xAccidOn:=xAccidIsGoing3 );

AccidAlkaliSwitch_4(
	xV_AccidOut:= xState_V403,
	xV_AlkaliOut:= xState_V404,
	xAccidOn:=xAccidIsGoing4 );





Conc_Line_1(
	value:= AI_Conc_Line1,
	min_value:= ,
	max_value:= 999.9,
	crash_value_4_20ma_1:= , 
	crash_value_4_20ma_2:= ,
	value_int:= ,
	crash_value_PT100_1:= ,
	crash_value_PT100_2:= , 
	sensor_offset:= ,
	sensor_gain:= ,
	rezult_value=> Conc_Line1_raw,
	crash_value=> ,
	out_crash_int=> );

Conc_Line_2(
	value:= AI_Conc_Line2,
	min_value:= ,
	max_value:= 999.9,
	crash_value_4_20ma_1:= ,
	crash_value_4_20ma_2:= , 
	value_int:= , 
	crash_value_PT100_1:= ,
	crash_value_PT100_2:= , 
	sensor_offset:= ,
	sensor_gain:= , 
	rezult_value=> Conc_Line2_raw,
	crash_value=> , 
	out_crash_int=> );

Conc_Line_3(
	value:= AI_Conc_Line3,
	min_value:= ,
	max_value:= 999.9,
	crash_value_4_20ma_1:= , 
	crash_value_4_20ma_2:= , 
	value_int:= , 
	crash_value_PT100_1:= , 
	crash_value_PT100_2:= , 
	sensor_offset:= ,
	sensor_gain:= , 
	rezult_value=> Conc_Line3_raw,
	crash_value=> , 
	out_crash_int=> );

Conc_Line_4(
	value:=AI_Conc_Line4 ,
	min_value:= 0,
	max_value:= 999.9,
	crash_value_4_20ma_1:= , 
	crash_value_4_20ma_2:= ,
	value_int:= ,
	crash_value_PT100_1:= ,
	crash_value_PT100_2:= , 
	sensor_offset:= ,
	sensor_gain:= , 
	rezult_value=> Conc_Line4_raw,
	crash_value=> , 
	out_crash_int=> );


ConcEnd_Line_1(
	repair:= ,
	auto_status:= ,
	auto_mode:= ,
	xAccid:= xAccidIsGoing1,
	auto_cip_mode:= , 
	sensor_CT:= Conc_Line1_raw,
	sensor_temp:= Heater_BackTget_1,
	sensor_CT_error:= ,
	sensor_temp_error:= , 
	scheloch_b:= ,
	scheloch_d:= , 
	scheloch_f:= , 
	kislota_b:= ,
	kislota_d:= , 
	kislota_f:= ,
	choose_mode:= ,
	result=> Conc_Line1);

ConcEnd_Line_2(
	repair:= ,
	auto_status:= ,
	auto_mode:= ,
	xAccid:= xAccidIsGoing2,
	auto_cip_mode:= , 
	sensor_CT:= Conc_Line2_raw,
	sensor_temp:= Heater_BackTget_2,
	sensor_CT_error:= , 
	sensor_temp_error:= , 
	scheloch_b:= ,
	scheloch_d:= , 
	scheloch_f:= , 
	kislota_b:= , 
	kislota_d:= ,
	kislota_f:= , 
	choose_mode:= , 
	result=> Conc_Line2);

ConcEnd_Line_3(
	repair:= ,
	auto_status:= ,
	auto_mode:= ,
	xAccid:= xAccidIsGoing3,
	auto_cip_mode:= , 
	sensor_CT:= Conc_Line3_raw,
	sensor_temp:= Heater_BackTget_3,
	sensor_CT_error:= , 
	sensor_temp_error:= , 
	scheloch_b:= , 
	scheloch_d:= , 
	scheloch_f:= ,
	kislota_b:= ,
	kislota_d:= , 
	kislota_f:= , 
	choose_mode:= ,
	result=> Conc_Line3);

ConcEnd_Line_4(
	repair:= ,
	auto_status:= ,
	auto_mode:= ,
	xAccid:= xAccidIsGoing4,
	auto_cip_mode:= , 
	sensor_CT:= Conc_Line4_raw,
	sensor_temp:= Heater_BackTget_4,
	sensor_CT_error:= ,
	sensor_temp_error:= , 
	scheloch_b:= , 
	scheloch_d:= , 
	scheloch_f:= , 
	kislota_b:= , 
	kislota_d:= , 
	kislota_f:= ,
	choose_mode:= , 
	result=> Conc_Line4);
END_PROGRAM

(* POU Device/Sensors/fb_concentrator, ST *)
FUNCTION_BLOCK fb_concentrator
VAR_INPUT
	repair	:					BOOL	;
	auto_status	:			BOOL	;
	auto_mode	:			INT	;
	auto_cip_mode	:		INT	;
	sensor_CT	:			REAL	;
	sensor_temp	:			REAL	;
	sensor_CT_error	:		BOOL	;
	sensor_temp_error	:	BOOL	;
	scheloch_b	:			REAL:=2.5	;
	scheloch_d	:			REAL:=4.7	;
	scheloch_f	:			REAL:=0.018	;
	kislota_b	:				REAL:=2.7	;
	kislota_d	:				REAL:=5.4	;
	kislota_f	:				REAL:=0.017	;
	xAccid:						BOOL;
END_VAR

VAR_IN_OUT

	(*choose_mode:			INT;*)

END_VAR
VAR_OUTPUT
	result:						REAL;
END_VAR
VAR
	b	:						REAL	;
	d	:						REAL	;
	f	:						REAL	;
	choose_mode:			INT;

END_VAR
(*count concentration*)
IF repair = FALSE
THEN
    IF auto_status = TRUE AND auto_mode = 2
      THEN
        (*scheloch*)
        IF auto_cip_mode = 2 OR auto_cip_mode = 3 OR auto_cip_mode = 4
          THEN
            choose_mode:= 1;
        END_IF;
        (*kislota*)
        IF auto_cip_mode = 5 OR auto_cip_mode = 6 OR auto_cip_mode = 7
          THEN
            choose_mode:= 2;
        END_IF;
    END_IF;

    (*other choice*)
    IF choose_mode < 1 OR choose_mode > 2
      THEN
        choose_mode:= 1;
    END_IF;
    (*scheloch*)
    IF (*choose_mode = 1*)NOT xAccid
      THEN
        b:= scheloch_b;
        d:= scheloch_d;
        f:= scheloch_f;
    END_IF;
    (*kislota*)
    IF (*choose_mode = 2*)xAccid
      THEN
        b:= kislota_b;
        d:= kislota_d;
        f:= kislota_f;
    END_IF;

    (*count result*)
    IF ((2.0 * (d * f * sensor_temp - 20.0 * d * f + d)) <> 0) AND sensor_CT_error = FALSE AND sensor_temp_error = FALSE
      THEN
        result := (-2.0 * b * f * sensor_temp + d * f * sensor_temp + 40.0 * b * f - 20.0 * d * f + 2.0 * (sensor_CT / 10.0) - 2.0 * b + d) / (2.0 * (d * f * sensor_temp - 20.0 * d * f + d));
      ELSE
        result := 0;
    END_IF;
  ELSE
    result := 0;
END_IF;
END_FUNCTION_BLOCK

(* POU Device/Sensors/fbAccidAlkaliSwitch, ST *)
FUNCTION_BLOCK fbAccidAlkaliSwitch
VAR_INPUT
	xV_AccidOut:	BOOL;
	xV_AlkaliOut:	BOOL;
END_VAR
VAR_IN_OUT
	xAccidOn:		BOOL;
END_VAR
VAR_OUTPUT
END_VAR
VAR
	rtAccidOn:	R_TRIG;
	rtAlkaliOn:	R_TRIG;
END_VAR
rtAccidOn(CLK:=xV_AccidOut);
rtAlkaliOn(CLK:=xV_AlkaliOut);

IF(* rtAccidOn.Q*) xV_AccidOut THEN
	xAccidOn:=TRUE;
END_IF

IF (*rtAlkaliOn.Q*) xV_AlkaliOut THEN
	xAccidOn:=FALSE;
END_IF
END_FUNCTION_BLOCK

(* POU Device/Sensors/prLevel, ST *)
PROGRAM prLevel
VAR
	fbCleanWaterLeve: LIN_TRAFO;
	fbUsedWaterLeve: LIN_TRAFO;
	fbAccidLevel: LIN_TRAFO;
	fbAlkaliLevel: LIN_TRAFO;
	check: LIN_TRAFO;
	checkMax:REAL:=20;
	checkMin:REAL;
	OUT_MIN: REAL;
	OUT_MAX:REAL:=32765;

END_VAR
fbCleanWaterLeve(
	IN:= AI_CleanWaterLevel,
	IN_MIN:= 616,
	IN_MAX:= (*32762*)24540,
	OUT_MIN:= 0,
	OUT_MAX:= 100,
	ERROR=> );

	(*CleanWaterLevel:=fnPressureToVolume(fbCleanWaterLeve.OUT, 3.14);*)
	CleanWaterLevel:=fbCleanWaterLeve.OUT;
	IF AI_CleanWaterLevel> 24540 THEN
		CleanWaterLevel:= 101;
	END_IF

fbUsedWaterLeve(
	IN:= AI_UsedWaterLevel,
	IN_MIN:= 584,
	IN_MAX:= 24400,
	OUT_MIN:= 0,
	OUT_MAX:= 100,
	ERROR=> );

	(*UsedWaterLevel:=fnPressureToVolume(fbUsedWaterLeve.OUT, 3.14);*)
	UsedWaterLevel:=fbUsedWaterLeve.OUT;
	IF AI_UsedWaterLevel > 24400 THEN
		UsedWaterLevel:=101;
	END_IF

fbAccidLevel(
	IN:= AI_AccidLevel,
	IN_MIN:= 624,
	IN_MAX:= 24344,
	OUT_MIN:= 0,
	OUT_MAX:= 100,
	ERROR=> );

	(*AccidLevel:=fnPressureToVolume(fbAccidLevel.OUT, 3.14);*)
	AccidLevel:=fbAccidLevel.OUT;
	IF AI_AccidLevel > 24344 THEN
		AccidLevel:=101;
	END_IF

fbAlkaliLevel(
	IN:= AI_AlkaliLevel,
	IN_MIN:= 616,
	IN_MAX:= 24480,
	OUT_MIN:= 0,
	OUT_MAX:= 100,
	ERROR=> );

	(*AlkaliLevel:=fnPressureToVolume(fbAlkaliLevel.OUT, 3.14);*)
	AlkaliLevel:=fbAlkaliLevel.OUT;
	IF AI_AlkaliLevel > 24480 THEN
		AlkaliLevel:=101;
	END_IF

	check(
	IN:= 4.299,
	IN_MIN:= checkMin,
	IN_MAX:= checkMax,
	OUT_MIN:= OUT_MIN,
	OUT_MAX:= OUT_MAX,
	OUT=> , 
	ERROR=> );
(*

PRESSURE = (p * volume * g)/S

p = 0.998
g = 9.81

Volume = (PRESSURE * S)/(p * g)

*)
END_PROGRAM

(* POU Device/Sensors/prTemperature, ST *)
PROGRAM prTemperature
VAR
END_VAR
Temp_Accid	:=	WORD_TO_REAL(AI_Temp_Accid)/10;
Temp_Alkali	:=	WORD_TO_REAL(AI_Temp_Alkali)/10;
Temp_Line3	:=	WORD_TO_REAL(AI_Temp_Line3)/10;
Temp_Line4	:=	WORD_TO_REAL(AI_Temp_Line4)/10;
		
Heater_Tget_1 	:=	WORD_TO_REAL(AI_Heater_Tget_1 )/10;
Heater_Tget_2 	:=	WORD_TO_REAL(AI_Heater_Tget_2 )/10;
Heater_Tget_3 	:=	WORD_TO_REAL(AI_Heater_Tget_3 )/10;
Heater_Tget_4 	:=	WORD_TO_REAL(AI_Heater_Tget_4 )/10;
		
Heater_BackTget_1	:=	WORD_TO_REAL(AI_Heater_BackTget_1)/10;
Heater_BackTget_2	:=	WORD_TO_REAL(AI_Heater_BackTget_2)/10;
Heater_BackTget_3	:=	WORD_TO_REAL(AI_Heater_BackTget_3)/10;
Heater_BackTget_4	:=	WORD_TO_REAL(AI_Heater_BackTget_4)/10;


Temp_Accid	:=	WORD_TO_REAL(AI_Temp_Accid)/10;
Temp_Alkali	:=	WORD_TO_REAL(AI_Temp_Alkali)/10;
END_PROGRAM

(* POU Device/Heater/prHeater, ST *)
PROGRAM prHeater
VAR
	Heater_1:		fbHeater;
	Heater_2:		fbHeater;
	Heater_3:		fbHeater;
	Heater_4:		fbHeater;

END_VAR
Heater_1(
	xManualMode:= Heater_xManualMode_1,
	xNoFeedback:= Heater_xNoFeedback_1,
	wTautoSet:= Heater_AutoSetT_1,
	wPowerManualSet:= Heater_PowerSet_1,
	wKp:= Heater_Kp,
	wKi:= Heater_Ki,
	wKd:= Heater_Kd,
	wMaxPower:= Heater_wMaxPower,
	wMinPower:= Heater_wMinPower,
	wTget:= Heater_Tget_1,
	wFlawGet:= Pump_FlawGet_1,
	xPumpWorking:=Pump_FeedbackOn_1,
	xInterlock:= ,
	wTmanualSet:=Heater_ManualSetT_1,
	wAO_Power=> HeaterPowerSet_1,
	wError=> Heater_Error_1 );


Heater_2(
	xManualMode:= Heater_xManualMode_2,
	xNoFeedback:= Heater_xNoFeedback_2,
	wTautoSet:= Heater_AutoSetT_2,
	wPowerManualSet:= Heater_PowerSet_2,
	wKp:= Heater_Kp,
	wKi:= Heater_Ki,
	wKd:= Heater_Kd,
	wMaxPower:= Heater_wMaxPower,
	wMinPower:= Heater_wMinPower,
	wTget:= Heater_Tget_2,
	wFlawGet:= Pump_FlawGet_2,
	xPumpWorking:=Pump_FeedbackOn_2,
	xInterlock:= ,
	wTmanualSet:=Heater_ManualSetT_2,
	wAO_Power=> HeaterPowerSet_2,
	wError=> Heater_Error_2 );


Heater_3(
	xManualMode:= Heater_xManualMode_3,
	xNoFeedback:= Heater_xNoFeedback_3,
	wTautoSet:= Heater_AutoSetT_3,
	wPowerManualSet:= Heater_PowerSet_3,
	wKp:= Heater_Kp,
	wKi:= Heater_Ki,
	wKd:= Heater_Kd,
	wMaxPower:= Heater_wMaxPower,
	wMinPower:= Heater_wMinPower,
	wTget:= Heater_Tget_3,
	wFlawGet:= Pump_FlawGet_3,
	xPumpWorking:=Pump_FeedbackOn_3,
	xInterlock:= ,
	wTmanualSet:=Heater_ManualSetT_3,
	wAO_Power=> HeaterPowerSet_3,
	wError=> Heater_Error_3 );


Heater_4(
	xManualMode:= Heater_xManualMode_4,
	xNoFeedback:= Heater_xNoFeedback_4,
	wTautoSet:= Heater_AutoSetT_4,
	wPowerManualSet:= Heater_PowerSet_4,
	wKp:= Heater_Kp,
	wKi:= Heater_Ki,
	wKd:= Heater_Kd,
	wMaxPower:= Heater_wMaxPower,
	wMinPower:= Heater_wMinPower,
	wTget:= Heater_Tget_4,
	wFlawGet:= Pump_FlawGet_4,
	xPumpWorking:=Pump_FeedbackOn_4,
	xInterlock:= ,
	wTmanualSet:=Heater_ManualSetT_4,
	wAO_Power=> HeaterPowerSet_4,
	wError=> Heater_Error_4 );
END_PROGRAM

(* POU Device/Heater/fbHeater, ST *)
FUNCTION_BLOCK fbHeater
VAR_INPUT
	xManualMode:			BOOL;
	xNoFeedback:			BOOL;
	wTautoSet:			REAL;
	wPowerManualSet:	REAL;
	wKp:					REAL;
	wKi:					REAL;
	wKd:					REAL;
	wMaxPower:			WORD;
	wMinPower:			WORD;
	wTget:					REAL;
	wFlawGet:				REAL;
	xInterlock:				BOOL;
	xPumpWorking:		BOOL;
END_VAR
VAR_IN_OUT
	wTmanualSet:			REAL;
END_VAR
VAR_OUTPUT
	wAO_Power:			REAL;
	wError:					WORD;
END_VAR
VAR
	fbAutoPID:				fbPID;
	tnNoFlaw:				TON;
END_VAR
IF xManualMode THEN
	IF (wTmanualSet > 0 OR xNoFeedback) AND wError = 0 THEN
		fbAutoPID(
			ACTUAL:= wTget,
			SET_POINT:= wTmanualSet,
			KP:= wKp,
			TN:= wKi,
			TV:= wKd,
			Y_MANUAL:= wPowerManualSet,
			Y_OFFSET:= ,
			Y_MIN:= wMinPower,
			Y_MAX:= wMaxPower,
			MANUAL:= xNoFeedback,
			RESET:= ,
			Y=> ,
			LIMITS_ACTIVE=> ,
			OVERFLOW=> );
			wAO_Power:= fbAutoPID.Y;
	ELSE
		wAO_Power:=0;
	END_IF
ELSE
	wTmanualSet:=wTautoSet;
	IF wTautoSet > 0 AND wError = 0 THEN
		fbAutoPID(
			ACTUAL:= wTget,
			SET_POINT:= wTautoSet,
			KP:= wKp,
			TN:= wKi,
			TV:= wKd,
			Y_MANUAL:= ,
			Y_OFFSET:= ,
			Y_MIN:= wMinPower,
			Y_MAX:= wMaxPower,
			MANUAL:=FALSE ,
			RESET:= ,
			Y=> ,
			LIMITS_ACTIVE=> ,
			OVERFLOW=> );
			wAO_Power:= fbAutoPID.Y;
	ELSE
		wAO_Power:=0;
	END_IF
END_IF



tnNoFlaw(IN:=  (NOT xPumpWorking) OR (wFlawGet = 0), PT:=T#1s, Q=>wError.0);
(*
IF tnNoFlaw.Q THEN
	wError.0:=TRUE;
END_IF
*)
END_FUNCTION_BLOCK

(* POU _ExtraFB/ControlFB/fbPID, ST *)
FUNCTION_BLOCK fbPID
VAR_INPUT
	ACTUAL :REAL;		(* actual value, process variable *)
	SET_POINT:REAL;	(* desired value, set point *)
	KP:REAL;				(* proportionality const. (P)*)
	TN:REAL;				(* reset time (I) in sec *)
	TV:REAL;				(* rate time, derivative time (D) in sec*)
	Y_MANUAL:REAL;		(* Y is set to this value as long as MANUAL=TRUE *)
	Y_OFFSET:REAL;		(* offset for manipulated variable *)
	Y_MIN:REAL;			(* minimum value for manipulated variable *)
	Y_MAX:REAL;			(* maximum value for manipulated variable *)
	MANUAL:BOOL;		(* 	TRUE: manual: Y is not influenced by controller,
								FALSE: controller determines Y *)
	RESET:BOOL;			(* reset: set Y output to Y_OFFSET and reset integral part *)
END_VAR
VAR_OUTPUT
	Y:REAL;				(* manipulated variable, set value*)
	LIMITS_ACTIVE:BOOL:=FALSE;	(* true set value would exceed limits Y_MIN, Y_MAX *)
	OVERFLOW:BOOL:=FALSE;		(* overflow in integral part *)
END_VAR
VAR
	CLOCK:TON;
	I: INTEGRAL;
	D: DERIVATIVE;
	TMDIFF: DWORD;
	ERROR: REAL;
	INIT: BOOL:=TRUE;
	Y_ADDOFFSET: REAL;
	KPcopy:REAL;
	TNcopy:REAL;
	TVcopy:REAL;
	rIntermediateVar:REAL;
END_VAR
IF TN>0 AND KP<> 0 AND (NOT OVERFLOW OR RESET OR MANUAL) THEN
	ERROR := SET_POINT-ACTUAL;								(* Regeldifferenz *)

	IF RESET OR MANUAL OR INIT OR (KP<>KPcopy OR TN<>TNcopy OR TV<>TVcopy) THEN							(* Reset oder Handbetrieb *)
		I(RESET:=TRUE);
		D(RESET:=TRUE);
		OVERFLOW:=FALSE;
		LIMITS_ACTIVE:=FALSE;
		IF RESET OR INIT THEN
			Y := Y_OFFSET;
			INIT:=FALSE;
			Y_ADDOFFSET := 0;
		ELSIF MANUAL THEN
			Y := Y_MANUAL;
			rIntermediateVar:=I.OUT/TN+D.OUT*TV;
			Y_ADDOFFSET := Y_MANUAL-(Y_OFFSET+KP*(ERROR)+rIntermediateVar);
			(*Y_ADDOFFSET := Y_MANUAL-(Y_OFFSET+KP*(ERROR)+(I.OUT/TN+D.OUT*TV));*)
		ELSE
			Y_ADDOFFSET := Y - Y_OFFSET - KP*ERROR;
		END_IF
		TMDIFF:=0;
		CLOCK(IN:=FALSE);									(* Timer neu starten *)
		CLOCK(PT:=t#1h, IN:=TRUE);

		TNcopy := TN;
		TVcopy := TV;
		KPcopy := KP;
	ELSE
		CLOCK;												(* Timer abfragen *)
		TMDIFF:=TIME_TO_DWORD(CLOCK.ET);					(* Zeitdifferenz seit letztem Aufruf *)
	END_IF;

	IF TMDIFF>0 THEN
		CLOCK(IN:=FALSE);									(* Timer neu starten *)
		CLOCK(PT:=t#1h, IN:=TRUE);

		D(IN:=ERROR, TM:=TMDIFF, RESET:=FALSE);				(* Differential abschätzen *)
		I(IN:=ERROR, TM:=TMDIFF, RESET:=FALSE);				(* Integral abschätzen *)

		OVERFLOW := I.OVERFLOW;
		IF NOT OVERFLOW THEN
			Y:=Y_OFFSET+KP*(ERROR)+(I.OUT/TN+D.OUT*TV) + Y_ADDOFFSET;
			IF Y>1E30 OR Y<-1E30 THEN						(* Overflow steht bevor, darf aber eigentlich nicht passieren *)
				OVERFLOW:=TRUE;
			END_IF;

			LIMITS_ACTIVE:=FALSE;
			IF Y_MAX>Y_MIN AND Y>Y_MAX  THEN				(* Stellwert-Obergrenze ьberschritten *)
				LIMITS_ACTIVE:=TRUE;
				IF KP<>0 THEN
					I(IN:=(Y_MAX-Y)*TN/KP,TM:=1000,RESET:=FALSE);		(* Integral korrigieren *)
				END_IF
				Y:=Y_MAX;
			END_IF;
			IF Y_MAX>Y_MIN AND Y<Y_MIN THEN					(* Stellwert-Untergrenze unterschritten *)
				LIMITS_ACTIVE:=TRUE;
				IF KP<>0 THEN
					I(IN:=(Y_MIN-Y)*TN/KP,TM:=1000,RESET:=FALSE);		(* Integral korrigieren *)
				END_IF
				Y:=Y_MIN;
			END_IF;
		END_IF;
	ELSE
		CLOCK(PT:=t#1h,IN:=TRUE);
	END_IF;

END_IF;
END_FUNCTION_BLOCK

(* POU _ExtraFB/mathematical functions/INTEGRAL, ST *)
(* function block to approximate the integral of IN over the time *)
FUNCTION_BLOCK INTEGRAL
VAR_INPUT
	IN:REAL;						(* input variable *)
	TM:DWORD;					(* time since last call in msec *)
	RESET:BOOL;					(* reset: OUT is set to zero and OVERFLOW to false *)
END_VAR
VAR_OUTPUT
	OUT:REAL;					(* value of the integral *)
	OVERFLOW:BOOL:=FALSE;	(* overflow *)
END_VAR
VAR
END_VAR
IF RESET THEN
	OUT:=0;
	OVERFLOW:=FALSE;
ELSIF NOT OVERFLOW  THEN
	IF 1E38 - IN*TM < OUT OR -1E38 - IN*TM > OUT THEN
		OVERFLOW:=TRUE;
	ELSE
		OUT:=OUT+IN*TM/1000;
	END_IF;
END_IF;
END_FUNCTION_BLOCK

(* POU _ExtraFB/mathematical functions/DERIVATIVE, ST *)
(* function block to approximate the derivative of a value *)
(* to calculate this, always four values are used in order to be as exact as possible *)
FUNCTION_BLOCK DERIVATIVE
VAR_INPUT
	IN:REAL;						(* input variable *)
	TM:DWORD;					(* time since last call in msec *)
	RESET:BOOL;					(* reset: set OUT to zero *)
END_VAR
VAR_OUTPUT
	OUT:REAL;					(* derivative *)
END_VAR
VAR
	X3,X2,X1:REAL;
	T2,T1:DWORD;
	INIT:BOOL:=TRUE;
END_VAR
IF INIT OR RESET THEN
	X1:=IN;
	X2:=IN;
	X3:=IN;
	OUT:=0;
	INIT:=FALSE;
ELSE
	IF TM>0 THEN
		OUT:=(3*(IN-X3)+X1-X2)/((3*T2+4*T1+3*TM))*1000;
		X3:=X2;
		X2:=X1;
		X1:=IN;
		T2:=T1;
		T1:=TM;
	END_IF;
END_IF;
END_FUNCTION_BLOCK

(* POU Device/Pump/prPump, ST *)
PROGRAM prPump
VAR

	Pump_1:	fbPumpPID;
	Pump_2:	fbPumpPID;
	Pump_3:	fbPumpPID;
	Pump_4:	fbPumpPID;

	xResetErr: BOOL;

	PA1:		fbValve;
	PA2:		fbValve;
	PA3:		fbValve;
	PA4:		fbValve;
	PA11:		fbValve;
	PA12:		fbValve;

	tnOnRemotePump_1	:	TON;
	tnOnRemotePump_2	:	TON;
	tnOnRemotePump_3	:	TON;
	tnOnRemotePump_4	:	TON;

	tnOnRemotePump_1_1	:	TON;
	tnOnRemotePump_1_2	:	TON;
	tnOnRemotePump_1_3	:	TON;

	tnOffRemotePump_1_1	:	TON;
	tnOffRemotePump_1_2	:	TON;
	tnOffRemotePump_1_3	:	TON;

	tnOffRemotePump_1	:	TON;
	tnOffRemotePump_2	:	TON;
	tnOffRemotePump_3	:	TON;
	tnOffRemotePump_4	:	TON;

	rtOffRemotePomp1:	R_TRIG;
	rtOffRemotePomp2:	R_TRIG;

	rtOffRemotePomp1_1:	R_TRIG;
	rtOffRemotePomp1_2:	R_TRIG;
	rtOffRemotePomp1_3:	R_TRIG;


END_VAR
Pump_1(
	xManualMode:= Pump_ManualMode_1,
	xInRotationFlg:=Pump_FeedbackOn_1,
	xOnAuto:= Pump_OnAuto_1,
	xNoFeedback:= Pump_NoFeedback_1,
	wFlawAutoSet:= Pump_FlawAutoSet_1,
	wFlawManualSet:= Pump_FlawManualSet_1,
	wVelocitySet:= Pump_VelocitySet_1,
	wFlawGet:= Pump_FlawGet_1,
	wKp:= Pump_Kp,
	wKi:= Pump_Ki,
	wKd:= Pump_Kd,
	xInvertorNorm:= Pump_InvNorm_1,
	wMaxSpeed:= Pump_MaxSpeed,
	wMinSpeed:= Pump_MinSpeed,
	xOnManual:= Pump_OnManual_1,
	xResetErr:= xResetAlmAll,
	xDO_On=> DO_PumpOn_1,
	wState=>Pump_State_1,
	wAO_SpeedSet=> PumpSpeedSet_1,
	wError=> Pump_Error_1);


Pump_2(
	xManualMode:= Pump_ManualMode_2,
	xInRotationFlg:=Pump_FeedbackOn_2,
	xOnAuto:= Pump_OnAuto_2,
	xNoFeedback:= Pump_NoFeedback_2,
	wFlawAutoSet:= Pump_FlawAutoSet_2,
	wFlawManualSet:= Pump_FlawManualSet_2,
	wVelocitySet:= Pump_VelocitySet_2,
	wFlawGet:= Pump_FlawGet_2,
	wKp:= Pump_Kp,
	wKi:= Pump_Ki,
	wKd:= Pump_Kd,
	xInvertorNorm:= Pump_InvNorm_2,
	wMaxSpeed:= Pump_MaxSpeed,
	wMinSpeed:= Pump_MinSpeed,
	xOnManual:= Pump_OnManual_2,
	xResetErr:= xResetAlmAll,
	xDO_On=> DO_PumpOn_2,
	wState=>Pump_State_2,
	wAO_SpeedSet=> PumpSpeedSet_2,
	wError=> Pump_Error_2);


Pump_3(
	xManualMode:= Pump_ManualMode_3,
	xInRotationFlg:=Pump_FeedbackOn_3,
	xOnAuto:= Pump_OnAuto_3,
	xNoFeedback:= Pump_NoFeedback_3,
	wFlawAutoSet:= Pump_FlawAutoSet_3,
	wFlawManualSet:= Pump_FlawManualSet_3,
	wVelocitySet:= Pump_VelocitySet_3,
	wFlawGet:= Pump_FlawGet_3,
	wKp:= Pump_Kp,
	wKi:= Pump_Ki,
	wKd:= Pump_Kd,
	xInvertorNorm:= Pump_InvNorm_3,
	wMaxSpeed:= Pump_MaxSpeed,
	wMinSpeed:= Pump_MinSpeed,
	xOnManual:= Pump_OnManual_3,
	xResetErr:= xResetAlmAll,
	xDO_On=> DO_PumpOn_3,
	wState=>Pump_State_3,
	wAO_SpeedSet=> PumpSpeedSet_3,
	wError=> Pump_Error_3);


Pump_4(
	xManualMode:= Pump_ManualMode_4,
	xInRotationFlg:=Pump_FeedbackOn_4,
	xOnAuto:= Pump_OnAuto_4,
	xNoFeedback:= Pump_NoFeedback_4,
	wFlawAutoSet:= Pump_FlawAutoSet_4,
	wFlawManualSet:= Pump_FlawManualSet_4,
	wVelocitySet:= Pump_VelocitySet_4,
	wFlawGet:= Pump_FlawGet_4,
	wKp:= Pump_Kp,
	wKi:= Pump_Ki,
	wKd:= Pump_Kd,
	xInvertorNorm:= Pump_InvNorm_4,
	wMaxSpeed:= Pump_MaxSpeed,
	wMinSpeed:= Pump_MinSpeed,
	xOnManual:= Pump_OnManual_4,
	xResetErr:= xResetAlmAll,
	xDO_On=> DO_PumpOn_4,
	wState=>Pump_State_4,
	wAO_SpeedSet=> PumpSpeedSet_4,
	wError=> Pump_Error_4);


	PA1(
	xManualMode:= PA_ManualMode_1,
	xOnAuto:= PA_OnAuto_1,
	wOffDelay:= 0,
	xSensor:= DO_PA1,
	xOnManual:= PA_OnManual_1,
	xResetError:=xResetErr,
	xDO_On=> DO_PA1,
	xState=> PA_State_1);

	PA2(
	xManualMode:= PA_ManualMode_2,
	xOnAuto:= PA_OnAuto_2,
	wOffDelay:= 0,
	xSensor:= DO_PA2,
	xOnManual:= PA_OnManual_2,
	xResetError:=xResetErr,
	xDO_On=> DO_PA2,
	xState=> PA_State_2);

	PA3(
	xManualMode:= PA_ManualMode_3,
	xOnAuto:= PA_OnAuto_3,
	wOffDelay:= 0,
	xSensor:= DO_PA3,
	xOnManual:= PA_OnManual_3,
	xResetError:=xResetErr,
	xDO_On=> DO_PA3,
	xState=> PA_State_3);

	PA4(
	xManualMode:= PA_ManualMode_4,
	xOnAuto:= PA_OnAuto_4,
	wOffDelay:= 0,
	xSensor:= DO_PA4,
	xOnManual:= PA_OnManual_4,
	xResetError:=xResetErr,
	xDO_On=> DO_PA4,
	xState=> PA_State_4);

	PA11(
	xManualMode:= PA_ManualMode_11,
	xOnAuto:= PA_OnAuto_11,
	wOffDelay:= 0,
	xSensor:= DO_PA11,
	xOnManual:= PA_OnManual_11,
	xResetError:=xResetErr,
	xDO_On=> DO_PA11,
	xState=> PA_State_11);

	PA12(
	xManualMode:= PA_ManualMode_12,
	xOnAuto:= PA_OnAuto_12,
	wOffDelay:= 0,
	xSensor:= DO_PA12,
	xOnManual:= PA_OnManual_12,
	xResetError:=xResetErr,
	xDO_On=> DO_PA12,
	xState=> PA_State_12);


	tnOnRemotePump_1(IN:=DO_PumpOn_1 AND wWashingStateLine1 > 0,PT:=(WORD_TO_TIME(RemotePumpOnDelay)*1000));
	tnOnRemotePump_2(IN:=DO_PumpOn_2 AND wWashingStateLine2 > 0 AND (wChosenRecipeLine2 = 1 OR wChosenRecipeLine2 = 2 OR wChosenRecipeLine2 = 3) ,PT:=(WORD_TO_TIME(RemotePumpOnDelay)*1000));
	tnOnRemotePump_3(IN:=DO_PumpOn_3 AND wWashingStateLine3 > 0AND (wChosenRecipeLine3 = 1 OR wChosenRecipeLine3 = 2 OR wChosenRecipeLine3 = 3),PT:=(WORD_TO_TIME(RemotePumpOnDelay2)*1000));
	tnOnRemotePump_4(IN:=DO_PumpOn_4 AND wWashingStateLine4 > 0,PT:=(WORD_TO_TIME(RemotePumpOnDelay)*1000));

	tnOnRemotePump_1_1(IN:=DO_PumpOn_1 AND wWashingStateLine1 > 0 AND (wChosenRecipeLine1 = 1 OR wChosenRecipeLine1 = 2 (*OR wChosenRecipeLine1 = 3*)) ,PT:=(WORD_TO_TIME(wDissolvingPauseStateLine1)*1000));
	tnOnRemotePump_1_2(IN:=DO_PumpOn_2 AND wWashingStateLine2 > 0 AND (wChosenRecipeLine2 = 4 OR wChosenRecipeLine2 = 5 (*OR wChosenRecipeLine1 = 3*)) ,PT:=(WORD_TO_TIME(wDissolvingPauseStateLine2)*1000));
	tnOnRemotePump_1_3(IN:=DO_PumpOn_3 AND wWashingStateLine3 > 0 AND (wChosenRecipeLine3 = 4 OR wChosenRecipeLine3 = 5(* OR wChosenRecipeLine1 = 3*)) ,PT:=(WORD_TO_TIME(wDissolvingPauseStateLine3)*1000));

	tnOffRemotePump_1(IN:=NOT DO_PumpOn_1 ,PT:=(WORD_TO_TIME(RemotePumpOffDelay)*1000));
	tnOffRemotePump_2(IN:=NOT DO_PumpOn_2 ,PT:=(WORD_TO_TIME(RemotePumpOffDelay)*1000));
	tnOffRemotePump_3(IN:=NOT DO_PumpOn_3 ,PT:=(WORD_TO_TIME(RemotePumpOffDelay2)*1000));
	tnOffRemotePump_4(IN:=NOT DO_PumpOn_4 ,PT:=(WORD_TO_TIME(RemotePumpOffDelay)*1000));

	tnOffRemotePump_1_1(IN:=NOT DO_PumpOn_1 ,PT:=(WORD_TO_TIME(wWashingPauseStateLine1)*1000));
	tnOffRemotePump_1_2(IN:=NOT DO_PumpOn_2 ,PT:=(WORD_TO_TIME(wWashingPauseStateLine2)*1000));
	tnOffRemotePump_1_3(IN:=NOT DO_PumpOn_3 ,PT:=(WORD_TO_TIME(wWashingPauseStateLine3)*1000));


	(*IF tnOnRemotePump_1.Q THEN
		SwitchOnRemotePump_1:=TRUE;
	END_IF*)
	IF tnOnRemotePump_2.Q THEN
		SwitchOnRemotePump_1:=TRUE;
	END_IF
	IF tnOnRemotePump_3.Q THEN
		SwitchOnRemotePump_2:=TRUE;
	END_IF
	(*IF tnOnRemotePump_4.Q THEN
		SwitchOnRemotePump_4:=TRUE;
	END_IF*)

	IF tnOnRemotePump_1_1.Q THEN
		SwitchOnRemotePump_1_1:=TRUE;
	END_IF
	IF tnOnRemotePump_1_2.Q THEN
		SwitchOnRemotePump_1_2:=TRUE;
	END_IF
	IF tnOnRemotePump_1_3.Q THEN
		SwitchOnRemotePump_1_3:=TRUE;
	END_IF


	rtOffRemotePomp1(CLK:= tnOffRemotePump_2.Q);
	rtOffRemotePomp2(CLK:= tnOffRemotePump_3.Q);

	rtOffRemotePomp1_1(CLK:= tnOffRemotePump_1_1.Q);
	rtOffRemotePomp1_2(CLK:= tnOffRemotePump_1_2.Q);
	rtOffRemotePomp1_3(CLK:= tnOffRemotePump_1_3.Q);

	(*IF tnOffRemotePump_1.Q THEN
		SwitchOnRemotePump_1:=FALSE;
	END_IF*)
	IF rtOffRemotePomp1.Q THEN
		SwitchOnRemotePump_1:=FALSE;
	END_IF
	IF rtOffRemotePomp2.Q THEN
		SwitchOnRemotePump_2:=FALSE;
	END_IF
	(*IF tnOffRemotePump_4.Q THEN
		SwitchOnRemotePump_4:=FALSE;
	END_IF*)
	IF rtOffRemotePomp1_1.Q THEN
		SwitchOnRemotePump_1_1:=FALSE;
	END_IF
	IF rtOffRemotePomp1_2.Q THEN
		SwitchOnRemotePump_1_2:=FALSE;
	END_IF
	IF rtOffRemotePomp1_3.Q THEN
		SwitchOnRemotePump_1_3:=FALSE;
	END_IF
END_PROGRAM

(* POU Device/Pump/fbPumpPID, ST *)
FUNCTION_BLOCK fbPumpPID
VAR_INPUT
	xManualMode:			BOOL;
	xOnAuto:				BOOL;
	xInRotationFlg:		BOOL;

	xNoFeedback:			BOOL;
	wFlawAutoSet:		REAL;
	wFlawManualSet:		REAL;
	wVelocitySet:			REAL;
	wFlawGet:				REAL;
	wKp:					REAL;
	wKi:					REAL;
	wKd:					REAL;
	wMaxSpeed:			WORD;
	wMinSpeed:			WORD;

	xInvertorNorm:			BOOL;

	(*xInterlock:				BOOL;*)
END_VAR
VAR_IN_OUT

	xOnManual:			BOOL;
	xResetErr:				BOOL;

END_VAR
VAR_OUTPUT
	xDO_On:				BOOL;
	wAO_SpeedSet:		REAL;
	wError:					WORD;
	wState:				WORD;
END_VAR
VAR
	fbAutoPID:				fbPID;
	(*tnInterlockOn:			TON;*)
	tnNoFlaw:				TON;
	rSetPrm:				REAL;
	xSetManual:			BOOL;
	rtManual:				R_TRIG;
	rtAuto:					R_TRIG;
	ftManual:				F_TRIG;
	ftAuto:					F_TRIG;
	RESET: BOOL;
END_VAR
rtManual(CLK:=xOnManual);
rtAuto(CLK:= xOnAuto);
ftManual(CLK:=xOnManual);
ftAuto(CLK:= xOnAuto);

IF ftManual.Q OR ftAuto.Q THEN
	RESET:=TRUE;;
END_IF
IF rtManual.Q OR rtAuto.Q THEN
	RESET:=FALSE;
END_IF

IF xManualMode THEN

		fbAutoPID(
		ACTUAL:= wFlawGet,
		SET_POINT:= (*wFlawManualSet*)rSetPrm,
		KP:= wKp,
		TN:= wKi,
		TV:= wKd,
		Y_MANUAL:=  wVelocitySet,
		Y_OFFSET:= ,
		Y_MIN:= wMinSpeed,
		Y_MAX:= wMaxSpeed,
		MANUAL:= xNoFeedback,
		RESET:= RESET,
		Y=> ,
		LIMITS_ACTIVE=> , 
		OVERFLOW=> );
		(*RESET:=FALSE;*)
		wAO_SpeedSet:= fbAutoPID.Y;

	IF xOnManual AND wError = 0 THEN
		xDO_On:=TRUE;
		rSetPrm:=wFlawManualSet;
	ELSE
		wAO_SpeedSet:=0;
		rSetPrm:=0;
		xDO_On:= FALSE;
	END_IF

ELSE

	(*IF wFlawAutoSet > 0 THEN*)
		fbAutoPID(
		ACTUAL:= wFlawGet,
		SET_POINT:= (*wFlawAutoSet*)rSetPrm,
		KP:= wKp,
		TN:= wKi,
		TV:= wKd,
		Y_MANUAL:= ,
		Y_OFFSET:= ,
		Y_MIN:= wMinSpeed,
		Y_MAX:= wMaxSpeed,
		MANUAL:= FALSE,
		RESET:=RESET ,
		Y=> ,
		LIMITS_ACTIVE=> ,
		OVERFLOW=> );
		(*RESET:=FALSE;*)
		wAO_SpeedSet:= fbAutoPID.Y;
	(*ELSE
		wAO_SpeedSet:=0;
	END_IF*)
	IF xOnAuto AND wError = 0 THEN
		xDO_On:=TRUE;
		rSetPrm:=wFlawAutoSet;
	ELSE
		wAO_SpeedSet:=0;
		rSetPrm:=0;
		xDO_On:= FALSE;
	END_IF
	xOnManual:=xOnAuto;

END_IF




tnNoFlaw(IN:=xDO_On AND (wFlawGet = 0), PT:=T#300s, Q=>wError.0);


IF (xDO_On AND (NOT xInRotationFlg)) OR (xInRotationFlg AND (NOT xDO_On)) THEN
	wState:=1;
ELSIF xDO_On AND xInRotationFlg THEN
	wState:=2;
ELSIF NOT (xDO_On OR xInRotationFlg) THEN
	wState:=0;
END_IF

IF NOT xInvertorNorm THEN
	wError.1:=TRUE;
ELSE
	wError.1:=FALSE;
END_IF
IF xResetErr THEN

	wError:=0;
END_IF
(*
IF tnNoFlaw.Q THEN
	wError.0:=TRUE;
END_IF
*)
END_FUNCTION_BLOCK

(* POU Device/Valve/fbValve, ST *)
FUNCTION_BLOCK fbValve
VAR_INPUT
	xManualMode:			BOOL;
	xOnAuto:				BOOL;
	wOffDelay:				WORD:=3;
	xSensor:				BOOL;
	xInterlock:				BOOL;

END_VAR
VAR_IN_OUT

	xOnManual:			BOOL;
	xResetError:			BOOL;

END_VAR
VAR_OUTPUT
	xDO_On:				BOOL;
	xState:					BOOL;
	wError:					WORD;
END_VAR
VAR
	tfOffDelay:				TOF;
	xDO_OnOld:			BOOL;
	tnErrorNotOpen:		TON;
	tnErrorNotClosed:		TON;
	rtSwitchToManual:		R_TRIG;

END_VAR
rtSwitchToManual(CLK:=xManualMode);
IF rtSwitchToManual.Q THEN
	xOnManual:=xOnAuto;
END_IF

IF xManualMode THEN
	tfOffDelay(IN:=xOnManual, PT:= WORD_TO_TIME(wOffDelay * 1000), Q=>xDO_On);
ELSE
	xOnManual:=FALSE;
	tfOffDelay(IN:=xOnAuto, PT:= WORD_TO_TIME(wOffDelay * 1000), Q=>xDO_On);
END_IF
xState:=xSensor;

IF xInterlock THEN
	xDO_On:=FALSE;
END_IF

tnErrorNotOpen(IN:= xDO_On AND (NOT xSensor), PT:=t#15S);
tnErrorNotClosed(IN:= (NOT xDO_On) AND xSensor, PT:=t#15S);

IF tnErrorNotOpen.Q THEN
	wError.0:=TRUE;
END_IF
IF tnErrorNotClosed.Q THEN
	wError.1:=TRUE;
END_IF

IF xResetError THEN
	tnErrorNotOpen(IN:=FALSE);
	tnErrorNotClosed(IN:=FALSE);
	wError:=0;
END_IF



(*
IF xDO_OnOld <> xDO_On THEN
	tnDelayState(IN:=TRUE, PT:=T#3S);
	IF tnDelayState.Q THEN
		xState:= 		xDO_On;
		xDO_OnOld:=	xDO_On;
		tnDelayState(IN:=FALSE);
	END_IF
END_IF
*)
END_FUNCTION_BLOCK

(* POU Device/Valve/prValve, ST *)
PROGRAM prValve
VAR

	Valve_V101	:	fbValve;
	Valve_V102	:	fbValve;
	Valve_V103	:	fbValve;
	Valve_V104	:	fbValve;
	Valve_V105	:	fbValve;
	Valve_V106	:	fbValve;
	Valve_V107	:	fbValve;
	Valve_V108	:	fbValve;
	Valve_V109	:	fbValve;
	Valve_V110	:	fbValve;
	Valve_V111	:	fbValve;
	Valve_V201	:	fbValve;
	Valve_V202	:	fbValve;
	Valve_V203	:	fbValve;
	Valve_V204	:	fbValve;
	Valve_V205	:	fbValve;
	Valve_V206	:	fbValve;
	Valve_V207	:	fbValve;
	Valve_V208	:	fbValve;
	Valve_V209	:	fbValve;
	Valve_V210	:	fbValve;
	Valve_V211	:	fbValve;
	Valve_V301	:	fbValve;
	Valve_V302	:	fbValve;
	Valve_V303	:	fbValve;
	Valve_V304	:	fbValve;
	Valve_V305	:	fbValve;
	Valve_V306	:	fbValve;
	Valve_V307	:	fbValve;
	Valve_V308	:	fbValve;
	Valve_V309	:	fbValve;
	Valve_V310	:	fbValve;
	Valve_V311	:	fbValve;
	Valve_V401	:	fbValve;
	Valve_V402	:	fbValve;
	Valve_V403	:	fbValve;
	Valve_V404	:	fbValve;
	Valve_V405	:	fbValve;
	Valve_V406	:	fbValve;
	Valve_V407	:	fbValve;
	Valve_V408	:	fbValve;
	Valve_V409	:	fbValve;
	Valve_V410	:	fbValve;
	Valve_V411	:	fbValve;
	Valve_V501	:	fbValve;
	Valve_V510	:	fbValve;
	Valve_V511	:	fbValve;
	Valve_V512	:	fbValve;
	Valve_V513	:	fbValve;
	Valve_V514	:	fbValve;
	Valve_V515	:	fbValve;
	WaterSupplyValve:	fbWaterSupplyValve;


	xOnAutoWorking: BOOL;
	xResetErrorValves: BOOL;
END_VAR
xResetErrorValves:=xResetAlmAll;


Valve_V101
(xManualMode:= ManualMode_V101,
xSensor:=DI_V101,
xOnAuto:= OnAuto_V101,
xResetError:= xResetErrorValves,
 xOnManual:= OnManual_V101,
xDO_On=> DO_V101,
wError=> wAlm_V101,
xState=> xState_V101);

Valve_V102
(xManualMode:= ManualMode_V102,
xSensor:=DI_V102,
xOnAuto:= OnAuto_V102,
xResetError:= xResetErrorValves,
xOnManual:= OnManual_V102,
xDO_On=> DO_V102,
wError=> wAlm_V102,
xState=> xState_V102);

Valve_V103
(xManualMode:= ManualMode_V103,
xSensor:=DI_V103,
xOnAuto:= OnAuto_V103,
xResetError:= xResetErrorValves,
xOnManual:= OnManual_V103,
xDO_On=> DO_V103,
wError=> wAlm_V103,
xState=> xState_V103);

Valve_V104
(xManualMode:= ManualMode_V104,
xSensor:=DI_V104,
xOnAuto:= OnAuto_V104,
xResetError:= xResetErrorValves,
xOnManual:= OnManual_V104,
xDO_On=> DO_V104,
wError=> wAlm_V104,
xState=> xState_V104);

Valve_V105
(xManualMode:= ManualMode_V105,
xSensor:=DI_V105,
xOnAuto:= OnAuto_V105,
xResetError:= xResetErrorValves,
xOnManual:= OnManual_V105,
xDO_On=> DO_V105,
wError=> wAlm_V105,
xState=> xState_V105);

Valve_V106
(xManualMode:= ManualMode_V106,
xSensor:=DI_V106,
xInterlock:= DI_AlkaliUpperLevel,
xOnAuto:= OnAuto_V106,
xResetError:= xResetErrorValves,
 xOnManual:= OnManual_V106,
xDO_On=> DO_V106,
wError=> wAlm_V106,
xState=> xState_V106);

Valve_V107
(xManualMode:= ManualMode_V107,
xSensor:=DI_V107,
xInterlock:= DI_AccidUpperLevel,
xOnAuto:= OnAuto_V107,
xResetError:= xResetErrorValves,
xOnManual:= OnManual_V107,
xDO_On=> DO_V107,
wError=> wAlm_V107,
xState=> xState_V107);

Valve_V108
(xManualMode:= ManualMode_V108,
xSensor:=DI_V108,
xInterlock:= DI_UsedWaterUpperLevel,
xOnAuto:= OnAuto_V108,
xResetError:= xResetErrorValves,
xOnManual:= OnManual_V108,
xDO_On=> DO_V108,
wError=> wAlm_V108,
xState=> xState_V108);

Valve_V109
(xManualMode:= ManualMode_V109,
xSensor:=DI_V109,
xOnAuto:= OnAuto_V109,
wOffDelay:=1,
xResetError:= xResetErrorValves,
xOnManual:= OnManual_V109,
xDO_On=> DO_V109,
wError=> wAlm_V109,
xState=> xState_V109);

Valve_V110
(xManualMode:= ManualMode_V110,
xSensor:=DI_V110,
xOnAuto:= OnAuto_V110,
xResetError:= xResetErrorValves,
 xOnManual:= OnManual_V110,
xDO_On=> DO_V110,
wError=> wAlm_V110,
xState=> xState_V110);

Valve_V111
(xManualMode:= ManualMode_V111,
xSensor:=DI_V111,
xOnAuto:= OnAuto_V111,
xResetError:= xResetErrorValves,
xOnManual:= OnManual_V111,
xDO_On=> DO_V111,
wError=> wAlm_V111,
xState=> xState_V111);

Valve_V201
(xManualMode:= ManualMode_V201,
xSensor:=DI_V201,
xOnAuto:= OnAuto_V201,
xResetError:= xResetErrorValves,
 xOnManual:= OnManual_V201,
xDO_On=> DO_V201,
wError=> wAlm_V201,
xState=> xState_V201);

Valve_V202
(xManualMode:= ManualMode_V202,
xSensor:=DI_V202,
xOnAuto:= OnAuto_V202,
xResetError:= xResetErrorValves,
xOnManual:= OnManual_V202,
xDO_On=> DO_V202,
wError=> wAlm_V202,
xState=> xState_V202);

Valve_V203
(xManualMode:= ManualMode_V203,
xSensor:=DI_V203,
xOnAuto:= OnAuto_V203,
xResetError:= xResetErrorValves,
xOnManual:= OnManual_V203,
xDO_On=> DO_V203,
wError=> wAlm_V203,
xState=> xState_V203);

Valve_V204
(xManualMode:= ManualMode_V204,
xSensor:=DI_V204,
xOnAuto:= OnAuto_V204,
xResetError:= xResetErrorValves,
xOnManual:= OnManual_V204,
xDO_On=> DO_V204,
wError=> wAlm_V204,
xState=> xState_V204);

Valve_V205
(xManualMode:= ManualMode_V205,
xSensor:=DI_V205,
xOnAuto:= OnAuto_V205,
xResetError:= xResetErrorValves,
 xOnManual:= OnManual_V205,
xDO_On=> DO_V205,
wError=> wAlm_V205,
xState=> xState_V205);

Valve_V206
(xManualMode:= ManualMode_V206,
xSensor:=DI_V206,
xInterlock:= DI_AlkaliUpperLevel,
xOnAuto:= OnAuto_V206,
xResetError:= xResetErrorValves,
xOnManual:= OnManual_V206,
xDO_On=> DO_V206,
wError=> wAlm_V206,
xState=> xState_V206);

Valve_V207
(xManualMode:= ManualMode_V207,
xSensor:=DI_V207,
xInterlock:= DI_AccidUpperLevel,
xOnAuto:= OnAuto_V207,
xResetError:= xResetErrorValves,
xOnManual:= OnManual_V207,
xDO_On=> DO_V207,
wError=> wAlm_V207,
xState=> xState_V207);

Valve_V208
(xManualMode:= ManualMode_V208,
xSensor:=DI_V208,
xInterlock:= DI_UsedWaterUpperLevel,
xOnAuto:= OnAuto_V208,
xResetError:= xResetErrorValves,
xOnManual:= OnManual_V208,
xDO_On=> DO_V208,
wError=> wAlm_V208,
xState=> xState_V208);

Valve_V209
(xManualMode:= ManualMode_V209,
xSensor:=DI_V209,
wOffDelay:=1,
xOnAuto:= OnAuto_V209,
xResetError:= xResetErrorValves,
xOnManual:= OnManual_V209,
xDO_On=> DO_V209,
wError=> wAlm_V209,
xState=> xState_V209);

Valve_V210
(xManualMode:= ManualMode_V210,
xSensor:=DI_V210,
xOnAuto:= OnAuto_V210,
xResetError:= xResetErrorValves,
xOnManual:= OnManual_V210,
xDO_On=> DO_V210,
wError=> wAlm_V210,
xState=> xState_V210);

Valve_V211
(xManualMode:= ManualMode_V211,
xSensor:=DI_V211,
xOnAuto:= OnAuto_V211,
xResetError:= xResetErrorValves,
xOnManual:= OnManual_V211,
xDO_On=> DO_V211,
wError=> wAlm_V211,
xState=> xState_V211);

Valve_V301
(xManualMode:= ManualMode_V301,
xSensor:=DI_V301,
xOnAuto:= OnAuto_V301,
xResetError:= xResetErrorValves,
xOnManual:= OnManual_V301,
xDO_On=> DO_V301,
wError=> wAlm_V301,
xState=> xState_V301);

Valve_V302
(xManualMode:= ManualMode_V302,
xSensor:=DI_V302,
xOnAuto:= OnAuto_V302,
xResetError:= xResetErrorValves,
xOnManual:= OnManual_V302,
xDO_On=> DO_V302,
wError=> wAlm_V302,
xState=> xState_V302);

Valve_V303
(xManualMode:= ManualMode_V303,
xSensor:=DI_V303,
xOnAuto:= OnAuto_V303,
xResetError:= xResetErrorValves,
 xOnManual:= OnManual_V303,
xDO_On=> DO_V303,
wError=> wAlm_V303,
xState=> xState_V303);

Valve_V304
(xManualMode:= ManualMode_V304,
xSensor:=DI_V304,
xOnAuto:= OnAuto_V304,
xResetError:= xResetErrorValves,
 xOnManual:= OnManual_V304,
xDO_On=> DO_V304,
wError=> wAlm_V304,
xState=> xState_V304);

Valve_V305
(xManualMode:= ManualMode_V305,
xSensor:=DI_V305,
xOnAuto:= OnAuto_V305,
xResetError:= xResetErrorValves,
xOnManual:= OnManual_V305,
xDO_On=> DO_V305,
wError=> wAlm_V305,
xState=> xState_V305);

Valve_V306
(xManualMode:= ManualMode_V306,
xSensor:=DI_V306,
xInterlock:= DI_AlkaliUpperLevel,
xOnAuto:= OnAuto_V306,
xResetError:= xResetErrorValves,
xOnManual:= OnManual_V306,
xDO_On=> DO_V306,
wError=> wAlm_V306,
xState=> xState_V306);

Valve_V307
(xManualMode:= ManualMode_V307,
xSensor:=DI_V307,
xInterlock:= DI_AccidUpperLevel,
xOnAuto:= OnAuto_V307,
xResetError:= xResetErrorValves,
xOnManual:= OnManual_V307,
xDO_On=> DO_V307,
wError=> wAlm_V307,
xState=> xState_V307);

Valve_V308
(xManualMode:= ManualMode_V308,
xSensor:=DI_V308,
wOffDelay:=1,
xInterlock:= DI_UsedWaterUpperLevel,
xOnAuto:= OnAuto_V308,
xResetError:= xResetErrorValves,
xOnManual:= OnManual_V308,
xDO_On=> DO_V308,
wError=> wAlm_V308,
xState=> xState_V308);

Valve_V309
(xManualMode:= ManualMode_V309,
xSensor:=DI_V309,
xOnAuto:= OnAuto_V309,
xResetError:= xResetErrorValves,
xOnManual:= OnManual_V309,
xDO_On=> DO_V309,
wError=> wAlm_V309,
xState=> xState_V309);

Valve_V310
(xManualMode:= ManualMode_V310,
xSensor:=DI_V310,
xOnAuto:= OnAuto_V310,
xResetError:= xResetErrorValves,
xOnManual:= OnManual_V310,
xDO_On=> DO_V310,
wError=> wAlm_V310,
xState=> xState_V310);

Valve_V311
(xManualMode:= ManualMode_V311,
xSensor:=DI_V311,
xOnAuto:= OnAuto_V311,
xResetError:= xResetErrorValves,
xOnManual:= OnManual_V311,
xDO_On=> DO_V311,
wError=> wAlm_V311,
xState=> xState_V311);

Valve_V401
(xManualMode:= ManualMode_V401,
xSensor:=DI_V401,
xOnAuto:= OnAuto_V401,
xResetError:= xResetErrorValves,
xOnManual:= OnManual_V401,
xDO_On=> DO_V401,
wError=> wAlm_V401,
xState=> xState_V401);

Valve_V402
(xManualMode:= ManualMode_V402,
xSensor:=DI_V402,
xOnAuto:= OnAuto_V402,
xResetError:= xResetErrorValves,
xOnManual:= OnManual_V402,
xDO_On=> DO_V402,
wError=> wAlm_V402,
xState=> xState_V402);

Valve_V403
(xManualMode:= ManualMode_V403,
xSensor:=DI_V403,
xOnAuto:= OnAuto_V403,
xResetError:= xResetErrorValves,
xOnManual:= OnManual_V403,
xDO_On=> DO_V403,
wError=> wAlm_V403,
xState=> xState_V403);

Valve_V404
(xManualMode:= ManualMode_V404,
xSensor:=DI_V404,
xOnAuto:= OnAuto_V404,
xResetError:= xResetErrorValves,
xOnManual:= OnManual_V404,
xDO_On=> DO_V404,
wError=> wAlm_V404,
xState=> xState_V404);

Valve_V405
(xManualMode:= ManualMode_V405,
xSensor:=DI_V405,
xOnAuto:= OnAuto_V405,
xResetError:= xResetErrorValves,
 xOnManual:= OnManual_V405,
xDO_On=> DO_V405,
wError=> wAlm_V405,
xState=> xState_V405);

Valve_V406
(xManualMode:= ManualMode_V406,
xSensor:=DI_V406,
xInterlock:= DI_AlkaliUpperLevel,
xOnAuto:= OnAuto_V406,
xResetError:= xResetErrorValves,
xOnManual:= OnManual_V406,
xDO_On=> DO_V406,
wError=> wAlm_V406,
xState=> xState_V406);

Valve_V407
(xManualMode:= ManualMode_V407,
xSensor:=DI_V407,
xInterlock:= DI_AccidUpperLevel,
xOnAuto:= OnAuto_V407,
xResetError:= xResetErrorValves,
xOnManual:= OnManual_V407,
xDO_On=> DO_V407,
wError=> wAlm_V407,
xState=> xState_V407);

Valve_V408
(xManualMode:= ManualMode_V408,
xSensor:=DI_V408,
xInterlock:= DI_UsedWaterUpperLevel,
xOnAuto:= OnAuto_V408,
xResetError:= xResetErrorValves,
xOnManual:= OnManual_V408,
xDO_On=> DO_V408,
wError=> wAlm_V408,
xState=> xState_V408);

Valve_V409
(xManualMode:= ManualMode_V409,
xSensor:=DI_V409,
wOffDelay:=1,
xOnAuto:= OnAuto_V409,
xResetError:= xResetErrorValves,
xOnManual:= OnManual_V409,
xDO_On=> DO_V409,
wError=> wAlm_V409,
xState=> xState_V409);

Valve_V410
(xManualMode:= ManualMode_V410,
xSensor:=DI_V410,
xOnAuto:= OnAuto_V410,
xResetError:= xResetErrorValves,
xOnManual:= OnManual_V410,
xDO_On=> DO_V410,
wError=> wAlm_V410,
xState=> xState_V410);

Valve_V411
(xManualMode:= ManualMode_V411,
xSensor:=DI_V411,
xOnAuto:= OnAuto_V411,
xResetError:= xResetErrorValves,
xOnManual:= OnManual_V411,
xDO_On=> DO_V411,
wError=> wAlm_V411,
xState=> xState_V411);

Valve_V510
(xManualMode:= ManualMode_V510,
xSensor:=DI_V510,
xOnAuto:= OnAuto_V510,
xResetError:= xResetErrorValves,
xOnManual:= OnManual_V510,
xDO_On=> DO_V510,
wError=> wAlm_V510,
xState=> xState_V510);

Valve_V511
(xManualMode:= ManualMode_V511,
xSensor:=DI_V511,
xOnAuto:= OnAuto_V511,
xResetError:= xResetErrorValves,
xOnManual:= OnManual_V511,
xDO_On=> DO_V511,
wError=> wAlm_V511,
xState=> xState_V511);

Valve_V512
(xManualMode:= ManualMode_V512,
xSensor:=DI_V512,
xOnAuto:= OnAuto_V512,
xResetError:= xResetErrorValves,
xOnManual:= OnManual_V512,
xDO_On=> DO_V512,
wError=> wAlm_V512,
xState=> xState_V512);

Valve_V513
(xManualMode:= ManualMode_V513,
xSensor:=DI_V513,
xOnAuto:= OnAuto_V513,
xResetError:= xResetErrorValves,
xOnManual:= OnManual_V513,
xDO_On=> DO_V513,
wError=> wAlm_V513,
xState=> xState_V513);

Valve_V514
(xManualMode:= ManualMode_V514,
xSensor:=DI_V514,
xOnAuto:= OnAuto_V514,
xResetError:= xResetErrorValves,
xOnManual:= OnManual_V514,
xDO_On=> DO_V514,
wError=> wAlm_V514,
xState=> xState_V514);

Valve_V515
(xManualMode:= ManualMode_V515,
xSensor:=DI_V515,
xOnAuto:= OnAuto_V515,
xResetError:= xResetErrorValves,
xOnManual:= OnManual_V515,
xDO_On=> DO_V515,
wError=> wAlm_V515,
xState=> xState_V515);



